C01810=1037.433,142.300,402.252,169.804,40.880,157.706
C01811=1037.427,142.051,402.274,169.802,40.880,157.706
C01812=1037.421,141.802,402.296,169.800,40.880,157.706
C01813=1037.415,141.552,402.317,169.797,40.880,157.706
C01814=1037.405,141.155,402.352,169.794,40.880,157.705
C01815=1037.395,140.757,402.386,169.790,40.881,157.705
C01816=1037.385,140.358,402.420,169.787,40.880,157.705
C01817=1037.376,139.961,402.454,169.783,40.880,157.705
C01818=1037.370,139.712,402.475,169.781,40.880,157.705
C01819=1037.363,139.462,402.497,169.777,40.880,157.704
C01820=1037.358,139.214,402.518,169.775,40.880,157.704
C01821=1037.352,138.965,402.540,169.773,40.880,157.704
C01822=1037.345,138.716,402.561,169.771,40.880,157.704
C01823=1037.339,138.467,402.583,169.768,40.880,157.704
C01824=1037.333,138.218,402.604,169.766,40.880,157.704
C01825=1037.327,137.968,402.625,169.764,40.880,157.704
C01826=1037.320,137.719,402.646,169.761,40.880,157.704
C01827=1037.315,137.471,402.667,169.759,40.880,157.704
C01828=1037.309,137.222,402.689,169.757,40.880,157.704
C01829=1037.302,136.973,402.710,169.754,40.880,157.703
C01830=1037.296,136.724,402.731,169.751,40.880,157.703
C01831=1037.290,136.474,402.752,169.749,40.881,157.703
C01832=1037.284,136.225,402.774,169.747,40.880,157.703
C01833=1037.277,135.976,402.795,169.744,40.881,157.703
C01834=1037.268,135.591,402.827,169.741,40.880,157.703
C01835=1037.259,135.205,402.861,169.737,40.881,157.703
C01836=1037.249,134.820,402.893,169.734,40.880,157.702
C01837=1037.240,134.434,402.925,169.730,40.881,157.702
C01838=1037.234,134.185,402.947,169.727,40.880,157.702
C01839=1037.227,133.936,402.968,169.725,40.881,157.702
C01840=1037.221,133.687,402.989,169.723,40.881,157.702
C01841=1037.215,133.438,403.010,169.720,40.881,157.702
C01842=1037.209,133.189,403.031,169.718,40.881,157.702
C01843=1037.203,132.940,403.052,169.716,40.881,157.702
C01844=1037.196,132.691,403.073,169.714,40.881,157.701
C01845=1037.190,132.441,403.094,169.711,40.881,157.701
C01846=1037.185,132.193,403.116,169.709,40.881,157.701
C01847=1037.178,131.943,403.136,169.707,40.881,157.701
C01848=1037.172,131.695,403.157,169.705,40.881,157.701
C01849=1037.166,131.446,403.179,169.703,40.881,157.701
C01850=1037.160,131.196,403.199,169.700,40.881,157.701
C01851=1037.154,130.948,403.220,169.698,40.881,157.701
C01852=1037.148,130.698,403.241,169.696,40.881,157.701
C01853=1037.141,130.449,403.262,169.693,40.881,157.700
C01854=1037.135,130.200,403.282,169.690,40.881,157.700
C01855=1037.129,129.951,403.303,169.688,40.882,157.700
C01856=1037.123,129.702,403.324,169.686,40.882,157.700
C01857=1037.116,129.453,403.345,169.683,40.882,157.700
C01858=1037.110,129.204,403.365,169.681,40.882,157.700
C01859=1037.104,128.955,403.387,169.679,40.882,157.700
C01860=1037.098,128.706,403.407,169.677,40.882,157.700
C01861=1037.091,128.457,403.428,169.674,40.883,157.700
C01862=1037.085,128.208,403.448,169.672,40.883,157.700
C01863=1037.079,127.958,403.469,169.670,40.883,157.700
C01864=1037.073,127.710,403.489,169.668,40.883,157.700
C01865=1037.067,127.460,403.510,169.665,40.883,157.699
C01866=1037.060,127.211,403.531,169.663,40.883,157.699
C01867=1037.054,126.962,403.551,169.661,40.884,157.699
C01868=1037.048,126.713,403.573,169.659,40.884,157.699
C01869=1037.042,126.464,403.593,169.655,40.883,157.699
C01870=1037.035,126.215,403.613,169.653,40.884,157.699
C01871=1037.029,125.967,403.634,169.651,40.884,157.699
C01872=1037.023,125.717,403.655,169.649,40.884,157.699
C01873=1037.016,125.467,403.675,169.646,40.884,157.699
C01874=1037.009,125.182,403.699,169.644,40.884,157.699
C01875=1037.002,124.897,403.723,169.641,40.884,157.699
C01876=1036.995,124.611,403.746,169.639,40.885,157.698
C01877=1036.988,124.325,403.770,169.636,40.885,157.698
C01878=1036.982,124.076,403.790,169.634,40.885,157.698
C01879=1036.976,123.826,403.811,169.632,40.885,157.698
C01880=1036.970,123.578,403.832,169.630,40.885,157.698
C01881=1036.963,123.329,403.852,169.627,40.885,157.698
C01882=1036.958,123.080,403.873,169.625,40.885,157.698
C01883=1036.951,122.831,403.894,169.623,40.885,157.698
C01884=1036.945,122.582,403.914,169.621,40.885,157.698
C01885=1036.938,122.332,403.934,169.619,40.886,157.698
C01886=1036.933,122.083,403.955,169.616,40.886,157.698
C01887=1036.926,121.834,403.976,169.613,40.886,157.697
C01888=1036.920,121.586,403.996,169.611,40.886,157.697
C01889=1036.914,121.336,404.016,169.609,40.886,157.697
C01890=1036.908,121.087,404.036,169.607,40.886,157.697
C01891=1036.902,120.839,404.057,169.604,40.886,157.697
C01892=1036.895,120.589,404.077,169.602,40.886,157.697
C01893=1036.890,120.340,404.098,169.600,40.886,157.697
C01894=1036.883,120.091,404.118,169.598,40.887,157.697
C01895=1036.877,119.842,404.138,169.596,40.887,157.697
C01896=1036.871,119.593,404.159,169.593,40.887,157.697
C01897=1036.865,119.344,404.180,169.591,40.887,157.696
C01898=1036.859,119.094,404.200,169.589,40.887,157.696
C01899=1036.853,118.845,404.220,169.587,40.887,157.696
C01900=1036.847,118.596,404.241,169.585,40.887,157.696
C01901=1036.841,118.347,404.261,169.581,40.887,157.696
C01902=1036.835,118.098,404.281,169.579,40.888,157.696
C01903=1036.828,117.849,404.302,169.577,40.888,157.696
C01904=1036.823,117.600,404.323,169.575,40.887,157.696
C01905=1036.817,117.351,404.343,169.573,40.888,157.696
C01906=1036.810,117.102,404.363,169.571,40.888,157.696
C01907=1036.804,116.853,404.383,169.568,40.888,157.696
C01908=1036.798,116.603,404.404,169.566,40.888,157.695
C01909=1036.792,116.354,404.424,169.564,40.888,157.695
C01910=1036.786,116.105,404.444,169.562,40.888,157.695
C01911=1036.780,115.856,404.464,169.560,40.888,157.695
C01912=1036.774,115.607,404.485,169.558,40.888,157.695
C01913=1036.768,115.358,404.504,169.556,40.888,157.695
C01914=1036.762,115.109,404.526,169.553,40.889,157.695
C01915=1036.756,114.860,404.545,169.550,40.888,157.695
C01916=1036.750,114.611,404.566,169.548,40.888,157.695
C01917=1036.744,114.362,404.586,169.546,40.889,157.695
C01918=1036.738,114.113,404.606,169.544,40.889,157.695
C01919=1036.732,113.864,404.626,169.542,40.888,157.694
C01920=1036.726,113.614,404.647,169.540,40.889,157.694
C01921=1036.720,113.365,404.667,169.537,40.889,157.694
C01922=1036.714,113.117,404.687,169.535,40.889,157.694
C01923=1036.707,112.867,404.707,169.533,40.889,157.694
C01924=1036.702,112.618,404.727,169.531,40.889,157.694
C01925=1036.696,112.369,404.747,169.529,40.889,157.694
C01926=1036.689,112.119,404.767,169.527,40.890,157.694
C01927=1036.683,111.870,404.787,169.524,40.890,157.694
C01928=1036.677,111.622,404.807,169.522,40.890,157.694
C01929=1036.670,111.372,404.827,169.520,40.890,157.694
C01930=1036.664,111.123,404.847,169.518,40.891,157.694
C01931=1036.659,110.874,404.866,169.516,40.890,157.693
C01932=1036.652,110.624,404.887,169.514,40.890,157.693
C01933=1036.646,110.376,404.907,169.511,40.891,157.693
C01934=1036.640,110.127,404.927,169.509,40.891,157.693
C01935=1036.633,109.878,404.946,169.507,40.891,157.693
C01936=1036.627,109.628,404.966,169.504,40.891,157.693
C01937=1036.621,109.379,404.986,169.502,40.892,157.693
C01938=1036.613,109.093,405.008,169.499,40.892,157.693
C01939=1036.606,108.807,405.031,169.497,40.892,157.693
C01940=1036.599,108.521,405.054,169.494,40.893,157.693
C01941=1036.592,108.236,405.077,169.492,40.893,157.693
C01942=1036.586,107.986,405.096,169.489,40.893,157.693
C01943=1036.579,107.738,405.116,169.487,40.893,157.693
C01944=1036.573,107.488,405.136,169.485,40.893,157.692
C01945=1036.567,107.239,405.155,169.483,40.893,157.692
C01946=1036.561,106.990,405.175,169.481,40.893,157.692
C01947=1036.555,106.741,405.195,169.479,40.894,157.692
C01948=1036.548,106.491,405.214,169.476,40.894,157.692
C01949=1036.542,106.243,405.234,169.474,40.894,157.692
C01950=1036.536,105.994,405.254,169.472,40.894,157.692
C01951=1036.530,105.744,405.274,169.470,40.895,157.692
C01952=1036.524,105.495,405.294,169.468,40.895,157.692
C01953=1036.517,105.246,405.313,169.466,40.895,157.692
C01954=1036.512,104.997,405.332,169.463,40.896,157.692
C01955=1036.505,104.747,405.353,169.461,40.896,157.692
C01956=1036.499,104.499,405.373,169.459,40.895,157.691
C01957=1036.493,104.249,405.392,169.457,40.896,157.691
C01958=1036.486,104.001,405.411,169.455,40.896,157.691
C01959=1036.481,103.751,405.431,169.453,40.896,157.691
C01960=1036.474,103.502,405.451,169.451,40.896,157.691
C01961=1036.468,103.253,405.471,169.448,40.897,157.691
C01962=1036.463,103.003,405.490,169.446,40.897,157.691
C01963=1036.456,102.755,405.509,169.443,40.897,157.691
C01964=1036.450,102.505,405.529,169.441,40.897,157.691
C01965=1036.444,102.256,405.549,169.439,40.897,157.691
C01966=1036.438,102.007,405.568,169.437,40.897,157.691
C01967=1036.432,101.758,405.588,169.435,40.897,157.691
C01968=1036.425,101.509,405.608,169.433,40.898,157.691
C01969=1036.419,101.260,405.627,169.430,40.898,157.691
C01970=1036.413,101.010,405.647,169.428,40.898,157.691
C01971=1036.407,100.761,405.666,169.426,40.898,157.690
C01972=1036.400,100.512,405.686,169.424,40.899,157.690
C01973=1036.395,100.263,405.705,169.422,40.898,157.690
C01974=1036.389,100.014,405.725,169.420,40.898,157.690
C01975=1036.382,99.765,405.744,169.418,40.899,157.690
C01976=1036.376,99.515,405.763,169.415,40.900,157.690
C01977=1036.369,99.266,405.783,169.413,40.900,157.690
C01978=1036.364,99.017,405.802,169.411,40.900,157.690
C01979=1036.357,98.768,405.821,169.409,40.900,157.690
C01980=1036.351,98.519,405.840,169.407,40.901,157.690
C01981=1036.344,98.269,405.859,169.405,40.901,157.690
C01982=1036.338,98.020,405.879,169.402,40.901,157.690
C01983=1036.332,97.771,405.898,169.400,40.901,157.690
C01984=1036.326,97.522,405.917,169.398,40.902,157.690
C01985=1036.319,97.273,405.937,169.396,40.902,157.690
C01986=1036.314,97.024,405.956,169.394,40.902,157.690
C01987=1036.307,96.774,405.975,169.392,40.902,157.689
C01988=1036.301,96.525,405.995,169.390,40.903,157.689
C01989=1036.294,96.276,406.014,169.387,40.903,157.689
C01990=1036.288,96.027,406.033,169.385,40.903,157.689
C01991=1036.282,95.778,406.052,169.383,40.903,157.689
C01992=1036.276,95.529,406.071,169.381,40.904,157.689
C01993=1036.270,95.280,406.090,169.379,40.904,157.689
C01994=1036.264,95.030,406.109,169.376,40.903,157.689
C01995=1036.257,94.781,406.129,169.374,40.904,157.689
C01996=1036.251,94.532,406.148,169.371,40.904,157.689
C01997=1036.244,94.282,406.167,169.369,40.904,157.689
C01998=1036.239,94.033,406.186,169.367,40.904,157.689
C01999=1036.232,93.785,406.206,169.365,40.905,157.689
C02000=1036.226,93.535,406.225,169.363,40.905,157.689
C02001=1036.220,93.286,406.243,169.361,40.905,157.688
C02002=1036.213,93.000,406.266,169.358,40.905,157.688
C02003=1036.205,92.714,406.287,169.356,40.906,157.688
C02004=1036.199,92.429,406.310,169.353,40.906,157.688
C02005=1036.192,92.142,406.332,169.351,40.906,157.688
C02006=1036.186,91.893,406.350,169.349,40.907,157.688
C02007=1036.180,91.644,406.369,169.347,40.907,157.688
C02008=1036.173,91.395,406.389,169.345,40.907,157.688
C02009=1036.168,91.146,406.408,169.343,40.907,157.688
C02010=1036.161,90.897,406.427,169.340,40.908,157.688
C02011=1036.155,90.648,406.445,169.338,40.908,157.688
C02012=1036.149,90.398,406.465,169.336,40.908,157.688
C02013=1036.143,90.149,406.483,169.334,40.908,157.688
C02014=1036.137,89.900,406.503,169.332,40.908,157.688
C02015=1036.130,89.651,406.522,169.330,40.909,157.688
C02016=1036.123,89.401,406.541,169.328,40.909,157.688
C02017=1036.117,89.152,406.560,169.325,40.909,157.687
C02018=1036.111,88.903,406.579,169.323,40.910,157.687
C02019=1036.105,88.654,406.597,169.321,40.910,157.687
C02020=1036.098,88.404,406.616,169.319,40.910,157.687
C02021=1036.092,88.155,406.635,169.317,40.910,157.687
C02022=1036.085,87.906,406.653,169.315,40.910,157.687
C02023=1036.080,87.657,406.673,169.313,40.911,157.687
C02024=1036.073,87.408,406.691,169.310,40.912,157.687
C02025=1036.067,87.159,406.710,169.308,40.912,157.687
C02026=1036.060,86.909,406.729,169.306,40.912,157.687
C02027=1036.054,86.660,406.747,169.304,40.912,157.687
C02028=1036.048,86.411,406.766,169.302,40.913,157.687
C02029=1036.042,86.161,406.784,169.300,40.913,157.687
C02030=1036.036,85.912,406.803,169.298,40.913,157.687
C02031=1036.029,85.663,406.822,169.295,40.913,157.687
C02032=1036.023,85.414,406.840,169.293,40.914,157.687
C02033=1036.017,85.164,406.860,169.291,40.914,157.687
C02034=1036.011,84.915,406.878,169.289,40.914,157.687
C02035=1036.004,84.666,406.897,169.286,40.914,157.686
C02036=1035.998,84.417,406.916,169.284,40.915,157.686
C02037=1035.992,84.168,406.934,169.282,40.915,157.686
C02038=1035.985,83.919,406.953,169.279,40.915,157.686
C02039=1035.979,83.669,406.972,169.278,40.916,157.686
C02040=1035.973,83.420,406.990,169.276,40.916,157.686
C02041=1035.967,83.170,407.009,169.273,40.916,157.686
C02042=1035.960,82.921,407.027,169.271,40.917,157.686
C02043=1035.954,82.672,407.046,169.269,40.917,157.686
C02044=1035.948,82.423,407.065,169.267,40.917,157.686
C02045=1035.942,82.174,407.084,169.265,40.917,157.686
C02046=1035.936,81.925,407.102,169.262,40.918,157.686
C02047=1035.930,81.675,407.120,169.260,40.918,157.686
C02048=1035.924,81.426,407.139,169.258,40.918,157.686
C02049=1035.917,81.177,407.157,169.256,40.918,157.686
C02050=1035.911,80.928,407.176,169.254,40.919,157.686
C02051=1035.905,80.679,407.195,169.252,40.919,157.686
C02052=1035.899,80.429,407.213,169.250,40.919,157.686
C02053=1035.892,80.180,407.232,169.248,40.919,157.686
C02054=1035.886,79.931,407.250,169.246,40.920,157.685
C02055=1035.880,79.682,407.269,169.243,40.920,157.685
C02056=1035.874,79.432,407.287,169.241,40.920,157.685
C02057=1035.868,79.183,407.306,169.239,40.920,157.685
C02058=1035.862,78.934,407.325,169.237,40.921,157.685
C02059=1035.856,78.685,407.343,169.235,40.921,157.685
C02060=1035.849,78.435,407.361,169.233,40.921,157.685
C02061=1035.843,78.186,407.380,169.231,40.921,157.685
C02062=1035.837,77.937,407.398,169.229,40.922,157.685
C02063=1035.830,77.687,407.416,169.226,40.922,157.685
C02064=1035.824,77.438,407.435,169.224,40.922,157.685
C02065=1035.818,77.190,407.453,169.222,40.922,157.685
C02066=1035.811,76.903,407.475,169.220,40.923,157.685
C02067=1035.804,76.617,407.495,169.217,40.924,157.685
C02068=1035.796,76.331,407.516,169.215,40.924,157.685
C02069=1035.790,76.046,407.537,169.212,40.924,157.685
C02070=1035.783,75.797,407.556,169.210,40.924,157.685
C02071=1035.777,75.547,407.574,169.208,40.925,157.684
C02072=1035.771,75.298,407.592,169.206,40.925,157.684
C02073=1035.764,75.048,407.610,169.204,40.925,157.684
C02074=1035.757,74.799,407.628,169.202,40.925,157.684
C02075=1035.751,74.549,407.646,169.200,40.926,157.684
C02076=1035.745,74.301,407.665,169.197,40.927,157.684
C02077=1035.739,74.051,407.683,169.195,40.927,157.684
C02078=1035.733,73.802,407.701,169.193,40.927,157.684
C02079=1035.727,73.553,407.720,169.191,40.927,157.684
C02080=1035.720,73.303,407.738,169.189,40.928,157.684
C02081=1035.713,73.054,407.756,169.187,40.928,157.684
C02082=1035.708,72.805,407.773,169.185,40.928,157.684
C02083=1035.701,72.556,407.792,169.182,40.928,157.684
C02084=1035.695,72.307,407.810,169.180,40.929,157.684
C02085=1035.689,72.057,407.829,169.178,40.929,157.684
C02086=1035.683,71.808,407.847,169.176,40.930,157.684
C02087=1035.677,71.559,407.864,169.174,40.930,157.684
C02088=1035.671,71.309,407.883,169.172,40.930,157.684
C02089=1035.664,71.060,407.900,169.170,40.930,157.684
C02090=1035.657,70.811,407.919,169.168,40.931,157.684
C02091=1035.651,70.561,407.937,169.165,40.931,157.683
C02092=1035.645,70.313,407.955,169.163,40.931,157.683
C02093=1035.639,70.063,407.973,169.161,40.931,157.683
C02094=1035.633,69.813,407.991,169.159,40.932,157.683
C02095=1035.626,69.564,408.009,169.157,40.933,157.683
C02096=1035.621,69.315,408.026,169.155,40.933,157.683
C02097=1035.614,69.066,408.045,169.153,40.933,157.683
C02098=1035.608,68.817,408.063,169.150,40.933,157.683
C02099=1035.601,68.567,408.080,169.148,40.934,157.683
C02100=1035.595,68.318,408.099,169.146,40.934,157.683
C02101=1035.589,68.069,408.117,169.144,40.934,157.683
C02102=1035.583,67.819,408.135,169.142,40.934,157.683
C02103=1035.576,67.570,408.153,169.140,40.935,157.683
C02104=1035.570,67.321,408.171,169.138,40.935,157.683
C02105=1035.564,67.072,408.188,169.135,40.936,157.683
C02106=1035.557,66.822,408.205,169.133,40.936,157.683
C02107=1035.551,66.573,408.224,169.131,40.936,157.683
C02108=1035.545,66.324,408.242,169.129,40.936,157.683
C02109=1035.539,66.075,408.259,169.127,40.937,157.683
C02110=1035.532,65.826,408.278,169.125,40.938,157.683
C02111=1035.526,65.576,408.296,169.123,40.938,157.683
C02112=1035.520,65.327,408.313,169.120,40.938,157.683
C02113=1035.514,65.077,408.330,169.118,40.938,157.683
C02114=1035.508,64.828,408.348,169.116,40.939,157.682
C02115=1035.501,64.579,408.366,169.114,40.939,157.682
C02116=1035.495,64.330,408.384,169.112,40.940,157.682
C02117=1035.488,64.080,408.401,169.110,40.940,157.682
C02118=1035.482,63.831,408.419,169.108,40.940,157.682
C02119=1035.476,63.581,408.437,169.105,40.940,157.682
C02120=1035.470,63.332,408.454,169.103,40.941,157.682
C02121=1035.462,63.083,408.472,169.101,40.942,157.682
C02122=1035.456,62.834,408.490,169.099,40.942,157.682
C02123=1035.450,62.585,408.507,169.097,40.942,157.682
C02124=1035.444,62.335,408.525,169.095,40.943,157.682
C02125=1035.437,62.086,408.542,169.092,40.943,157.682
C02126=1035.431,61.837,408.559,169.090,40.944,157.682
C02127=1035.425,61.587,408.577,169.088,40.944,157.682
C02128=1035.418,61.338,408.595,169.086,40.945,157.682
C02129=1035.411,61.088,408.612,169.084,40.945,157.682
C02130=1035.404,60.802,408.632,169.081,40.945,157.682
C02131=1035.397,60.516,408.652,169.079,40.946,157.682
C02132=1035.389,60.230,408.672,169.076,40.946,157.682
C02133=1035.382,59.944,408.692,169.074,40.947,157.682
C02134=1035.376,59.694,408.710,169.071,40.948,157.682
C02135=1035.369,59.446,408.727,169.069,40.948,157.682
C02136=1035.363,59.196,408.744,169.067,40.948,157.682
C02137=1035.356,58.947,408.762,169.065,40.948,157.682
C02138=1035.350,58.698,408.779,169.063,40.949,157.682
C02139=1035.344,58.448,408.797,169.060,40.950,157.682
C02140=1035.337,58.199,408.814,169.058,40.950,157.682
C02141=1035.331,57.950,408.831,169.056,40.950,157.682
C02142=1035.325,57.700,408.849,169.054,40.951,157.682
C02143=1035.318,57.451,408.866,169.052,40.951,157.682
C02144=1035.312,57.202,408.883,169.050,40.951,157.682
C02145=1035.305,56.952,408.901,169.047,40.952,157.681
C02146=1035.299,56.703,408.919,169.045,40.953,157.682
C02147=1035.292,56.454,408.935,169.043,40.953,157.681
C02148=1035.286,56.204,408.953,169.041,40.953,157.681
C02149=1035.280,55.956,408.970,169.039,40.953,157.681
C02150=1035.273,55.706,408.988,169.037,40.954,157.681
C02151=1035.267,55.456,409.005,169.034,40.955,157.681
C02152=1035.261,55.207,409.022,169.032,40.955,157.681
C02153=1035.254,54.958,409.039,169.030,40.955,157.681
C02154=1035.249,54.709,409.057,169.028,40.955,157.681
C02155=1035.242,54.459,409.074,169.026,40.956,157.681
C02156=1035.236,54.210,409.091,169.024,40.956,157.681
C02157=1035.229,53.961,409.109,169.021,40.957,157.681
C02158=1035.223,53.711,409.126,169.019,40.957,157.681
C02159=1035.217,53.462,409.143,169.017,40.957,157.681
C02160=1035.211,53.212,409.161,169.015,40.958,157.681
C02161=1035.204,52.963,409.178,169.013,40.958,157.681
C02162=1035.197,52.714,409.195,169.011,40.959,157.681
C02163=1035.192,52.464,409.212,169.008,40.959,157.681
C02164=1035.185,52.215,409.229,169.006,40.959,157.681
C02165=1035.179,51.966,409.246,169.004,40.960,157.681
C02166=1035.173,51.716,409.264,169.002,40.960,157.681
C02167=1035.167,51.468,409.281,169.000,40.960,157.681
C02168=1035.160,51.218,409.298,168.998,40.961,157.681
C02169=1035.155,50.969,409.315,168.995,40.961,157.681
C02170=1035.148,50.719,409.332,168.993,40.962,157.681
C02171=1035.142,50.471,409.349,168.991,40.962,157.681
C02172=1035.135,50.220,409.366,168.989,40.962,157.681
C02173=1035.129,49.971,409.384,168.987,40.963,157.680
C02174=1035.123,49.722,409.401,168.985,40.963,157.680
C02175=1035.116,49.473,409.418,168.982,40.963,157.680
C02176=1035.111,49.223,409.435,168.980,40.964,157.680
C02177=1035.104,48.974,409.452,168.978,40.964,157.680
C02178=1035.097,48.725,409.469,168.976,40.965,157.680
C02179=1035.092,48.475,409.486,168.974,40.965,157.680
C02180=1035.085,48.226,409.504,168.972,40.965,157.680
C02181=1035.079,47.977,409.521,168.969,40.965,157.680
C02182=1035.073,47.727,409.537,168.967,40.966,157.680
C02183=1035.067,47.478,409.555,168.965,40.966,157.680
C02184=1035.061,47.229,409.572,168.963,40.967,157.680
C02185=1035.054,46.979,409.588,168.961,40.967,157.680
C02186=1035.049,46.730,409.606,168.959,40.967,157.680
C02187=1035.042,46.481,409.623,168.957,40.967,157.680
C02188=1035.036,46.231,409.640,168.954,40.968,157.680
C02189=1035.029,45.982,409.657,168.952,40.969,157.680
C02190=1035.024,45.732,409.674,168.950,40.969,157.680
C02191=1035.018,45.483,409.691,168.948,40.969,157.680
C02192=1035.011,45.234,409.708,168.946,40.969,157.680
C02193=1035.005,44.985,409.724,168.944,40.970,157.680
C02194=1034.998,44.699,409.744,168.941,40.970,157.679
C02195=1034.991,44.411,409.764,168.939,40.970,157.679
C02196=1034.984,44.125,409.783,168.936,40.971,157.679
C02197=1034.977,43.839,409.803,168.934,40.971,157.679
C02198=1034.971,43.590,409.819,168.932,40.972,157.679
C02199=1034.964,43.340,409.837,168.929,40.972,157.679
C02200=1034.958,43.091,409.853,168.927,40.972,157.679
C02201=1034.951,42.841,409.870,168.925,40.972,157.679
C02202=1034.945,42.592,409.887,168.923,40.973,157.679
C02203=1034.940,42.343,409.904,168.921,40.974,157.679
C02204=1034.933,42.093,409.921,168.918,40.974,157.679
C02205=1034.927,41.844,409.938,168.916,40.974,157.679
C02206=1034.920,41.594,409.954,168.914,40.975,157.679
C02207=1034.914,41.345,409.971,168.912,40.975,157.679
C02208=1034.908,41.096,409.988,168.910,40.975,157.679
C02209=1034.902,40.846,410.004,168.907,40.976,157.679
C02210=1034.895,40.597,410.021,168.905,40.977,157.679
C02211=1034.889,40.348,410.037,168.903,40.977,157.679
C02212=1034.883,40.098,410.054,168.901,40.977,157.679
C02213=1034.877,39.849,410.071,168.899,40.977,157.679
C02214=1034.870,39.599,410.088,168.896,40.978,157.679
C02215=1034.864,39.350,410.105,168.894,40.979,157.679
C02216=1034.858,39.101,410.121,168.892,40.979,157.679
C02217=1034.851,38.851,410.137,168.890,40.979,157.679
C02218=1034.845,38.602,410.154,168.888,40.979,157.679
C02219=1034.839,38.353,410.171,168.886,40.980,157.679
C02220=1034.833,38.103,410.187,168.883,40.981,157.679
C02221=1034.826,37.854,410.204,168.881,40.981,157.678
C02222=1034.820,37.605,410.221,168.879,40.981,157.678
C02223=1034.814,37.355,410.237,168.877,40.982,157.678
C02224=1034.807,37.106,410.253,168.875,40.982,157.678
C02225=1034.801,36.857,410.270,168.872,40.982,157.678
C02226=1034.794,36.607,410.286,168.870,40.983,157.678
C02227=1034.788,36.358,410.303,168.868,40.984,157.678
C02228=1034.782,36.108,410.319,168.866,40.984,157.678
C02229=1034.775,35.858,410.335,168.863,40.985,157.678
C02230=1034.769,35.610,410.352,168.861,40.985,157.678
C02231=1034.763,35.360,410.368,168.859,40.985,157.678
C02232=1034.757,35.111,410.384,168.858,40.986,157.678
C02233=1034.750,34.861,410.400,168.855,40.987,157.678
C02234=1034.744,34.612,410.417,168.853,40.987,157.678
C02235=1034.737,34.363,410.434,168.851,40.988,157.678
C02236=1034.731,34.113,410.450,168.849,40.988,157.678
C02237=1034.724,33.864,410.466,168.846,40.988,157.678
C02238=1034.718,33.615,410.482,168.844,40.989,157.678
C02239=1034.712,33.365,410.499,168.842,40.989,157.678
C02240=1034.706,33.115,410.515,168.840,40.990,157.678
C02241=1034.700,32.866,410.531,168.838,40.990,157.678
C02242=1034.693,32.617,410.547,168.835,40.991,157.678
C02243=1034.686,32.368,410.564,168.833,40.991,157.678
C02244=1034.680,32.118,410.581,168.831,40.991,157.678
C02245=1034.674,31.869,410.597,168.829,40.992,157.678
C02246=1034.668,31.620,410.613,168.826,40.993,157.678
C02247=1034.662,31.371,410.629,168.824,40.993,157.678
C02248=1034.655,31.120,410.645,168.822,40.994,157.678
C02249=1034.649,30.871,410.662,168.820,40.994,157.678
C02250=1034.643,30.622,410.677,168.817,40.994,157.678
C02251=1034.637,30.373,410.694,168.815,40.995,157.678
C02252=1034.630,30.123,410.710,168.813,40.995,157.678
C02253=1034.623,29.874,410.726,168.811,40.996,157.678
C02254=1034.617,29.624,410.742,168.808,40.996,157.678
C02255=1034.611,29.375,410.758,168.806,40.997,157.678
C02256=1034.606,29.126,410.775,168.804,40.997,157.678
C02257=1034.598,28.876,410.791,168.802,40.997,157.677
C02258=1034.592,28.589,410.810,168.799,40.998,157.678
C02259=1034.584,28.303,410.829,168.797,40.999,157.677
C02260=1034.577,28.016,410.847,168.794,40.999,157.677
C02261=1034.570,27.730,410.865,168.791,41.000,157.677
C02262=1034.563,27.481,410.881,168.789,41.000,157.677
C02263=1034.557,27.232,410.897,168.787,41.000,157.677
C02264=1034.551,26.982,410.913,168.785,41.001,157.677
C02265=1034.544,26.733,410.929,168.782,41.002,157.677
C02266=1034.538,26.483,410.946,168.780,41.002,157.677
C02267=1034.531,26.233,410.961,168.778,41.003,157.677
C02268=1034.526,25.984,410.977,168.776,41.003,157.677
C02269=1034.519,25.735,410.992,168.773,41.004,157.677
C02270=1034.513,25.486,411.009,168.771,41.004,157.677
C02271=1034.506,25.237,411.024,168.769,41.004,157.677
C02272=1034.500,24.987,411.041,168.767,41.005,157.677
C02273=1034.493,24.737,411.056,168.764,41.006,157.677
C02274=1034.487,24.488,411.072,168.762,41.006,157.677
C02275=1034.481,24.239,411.088,168.761,41.007,157.677
C02276=1034.475,23.989,411.104,168.758,41.007,157.677
C02277=1034.468,23.740,411.120,168.756,41.008,157.677
C02278=1034.462,23.490,411.136,168.754,41.008,157.677
C02279=1034.455,23.241,411.151,168.752,41.008,157.677
C02280=1034.449,22.991,411.168,168.749,41.009,157.677
C02281=1034.442,22.742,411.183,168.747,41.010,157.677
C02282=1034.436,22.493,411.200,168.745,41.010,157.677
C02283=1034.430,22.243,411.214,168.743,41.011,157.677
C02284=1034.424,21.994,411.231,168.740,41.011,157.677
C02285=1034.417,21.745,411.246,168.738,41.011,157.677
C02286=1034.411,21.495,411.263,168.736,41.012,157.677
C02287=1034.405,21.246,411.278,168.733,41.013,157.677
C02288=1034.399,20.996,411.294,168.731,41.014,157.677
C02289=1034.392,20.747,411.310,168.729,41.014,157.677
C02290=1034.386,20.497,411.325,168.727,41.014,157.677
C02291=1034.380,20.248,411.341,168.724,41.015,157.677
C02292=1034.374,19.998,411.357,168.722,41.015,157.677
C02293=1034.367,19.749,411.372,168.720,41.015,157.677
C02294=1034.361,19.499,411.389,168.717,41.016,157.677
C02295=1034.355,19.250,411.404,168.715,41.017,157.677
C02296=1034.348,19.001,411.419,168.713,41.017,157.677
C02297=1034.342,18.751,411.435,168.711,41.018,157.677
C02298=1034.336,18.502,411.451,168.708,41.018,157.677
C02299=1034.329,18.253,411.466,168.706,41.019,157.677
C02300=1034.323,18.003,411.482,168.704,41.019,157.677
C02301=1034.317,17.754,411.497,168.701,41.020,157.677
C02302=1034.310,17.505,411.513,168.699,41.021,157.676
C02303=1034.304,17.255,411.528,168.697,41.021,157.676
C02304=1034.298,17.006,411.544,168.694,41.022,157.676
C02305=1034.290,16.756,411.560,168.692,41.022,157.676
C02306=1034.285,16.506,411.576,168.691,41.023,157.676
C02307=1034.278,16.257,411.591,168.688,41.023,157.676
C02308=1034.272,16.007,411.606,168.685,41.024,157.676
C02309=1034.266,15.758,411.623,168.684,41.024,157.676
C02310=1034.259,15.508,411.637,168.682,41.025,157.676
C02311=1034.253,15.259,411.653,168.679,41.025,157.676
C02312=1034.247,15.009,411.669,168.677,41.026,157.676
C02313=1034.240,14.760,411.684,168.675,41.026,157.676
C02314=1034.234,14.510,411.699,168.672,41.027,157.676
C02315=1034.228,14.261,411.716,168.670,41.027,157.676
C02316=1034.222,14.011,411.730,168.668,41.028,157.676
C02317=1034.215,13.762,411.746,168.665,41.029,157.676
C02318=1034.209,13.513,411.761,168.663,41.029,157.676
C02319=1034.202,13.263,411.776,168.661,41.030,157.676
C02320=1034.196,13.014,411.792,168.658,41.030,157.676
C02321=1034.190,12.764,411.807,168.656,41.031,157.676
C02322=1034.183,12.480,411.825,168.653,41.032,157.676
C02323=1034.175,12.194,411.842,168.651,41.032,157.676
C02324=1034.168,11.908,411.859,168.648,41.033,157.676
C02325=1034.161,11.623,411.877,168.645,41.034,157.676
C02326=1034.154,11.374,411.892,168.643,41.034,157.676
C02327=1034.148,11.125,411.907,168.640,41.035,157.676
C02328=1034.141,10.875,411.922,168.638,41.036,157.676
C02329=1034.135,10.625,411.937,168.636,41.036,157.676
C02330=1034.128,10.376,411.953,168.634,41.037,157.676
C02331=1034.122,10.127,411.968,168.632,41.037,157.676
C02332=1034.115,9.877,411.983,168.630,41.038,157.676
C02333=1034.109,9.629,411.998,168.627,41.038,157.676
C02334=1034.103,9.379,412.013,168.625,41.039,157.676
C02335=1034.097,9.129,412.028,168.623,41.040,157.676
C02336=1034.090,8.880,412.043,168.620,41.041,157.676
C02337=1034.083,8.631,412.059,168.618,41.041,157.676
C02338=1034.077,8.381,412.074,168.615,41.042,157.676
C02339=1034.071,8.131,412.089,168.613,41.042,157.676
C02340=1034.064,7.882,412.104,168.611,41.043,157.676
C02341=1034.058,7.632,412.119,168.608,41.043,157.676
C02342=1034.051,7.383,412.134,168.606,41.044,157.676
C02343=1034.045,7.133,412.149,168.604,41.044,157.676
C02344=1034.040,6.884,412.164,168.601,41.045,157.676
C02345=1034.033,6.634,412.179,168.599,41.046,157.676
C02346=1034.027,6.385,412.194,168.597,41.047,157.676
C02347=1034.020,6.136,412.210,168.594,41.047,157.676
C02348=1034.014,5.886,412.225,168.592,41.048,157.676
C02349=1034.008,5.636,412.240,168.589,41.048,157.676
C02350=1034.001,5.387,412.255,168.588,41.049,157.676
C02351=1033.995,5.138,412.269,168.585,41.049,157.676
C02352=1033.989,4.888,412.284,168.583,41.050,157.676
C02353=1033.982,4.639,412.300,168.581,41.051,157.676
C02354=1033.976,4.389,412.315,168.579,41.051,157.676
C02355=1033.970,4.140,412.330,168.576,41.052,157.676
C02356=1033.963,3.890,412.345,168.574,41.053,157.676
C02357=1033.957,3.641,412.359,168.571,41.053,157.676
C02358=1033.951,3.391,412.374,168.569,41.053,157.676
C02359=1033.945,3.142,412.389,168.567,41.054,157.676
C02360=1033.938,2.892,412.404,168.564,41.054,157.676
C02361=1033.932,2.642,412.419,168.562,41.055,157.676
C02362=1033.926,2.393,412.434,168.560,41.056,157.676
C02363=1033.920,2.144,412.449,168.557,41.057,157.676
C02364=1033.913,1.894,412.464,168.555,41.057,157.676
C02365=1033.907,1.645,412.478,168.552,41.058,157.676
C02366=1033.900,1.395,412.494,168.550,41.058,157.676
C02367=1033.894,1.147,412.509,168.548,41.058,157.676
C02368=1033.888,0.897,412.524,168.545,41.059,157.676
C02369=1033.882,0.647,412.539,168.543,41.060,157.676
C02370=1033.875,0.398,412.554,168.541,41.060,157.676
C02371=1033.870,0.149,412.568,168.538,41.061,157.676
C02372=1033.863,-0.101,412.583,168.536,41.062,157.676
C02373=1033.857,-0.351,412.598,168.533,41.062,157.675
C02374=1033.850,-0.600,412.613,168.531,41.062,157.675
C02375=1033.845,-0.850,412.627,168.529,41.063,157.675
C02376=1033.839,-1.100,412.642,168.526,41.064,157.675
C02377=1033.832,-1.349,412.657,168.525,41.064,157.675
C02378=1033.826,-1.598,412.671,168.523,41.065,157.675
C02379=1033.820,-1.848,412.686,168.520,41.066,157.675
C02380=1033.814,-2.098,412.701,168.518,41.066,157.675
C02381=1033.807,-2.347,412.716,168.515,41.066,157.675
C02382=1033.801,-2.596,412.731,168.513,41.067,157.675
C02383=1033.795,-2.846,412.746,168.511,41.067,157.675
C02384=1033.789,-3.095,412.761,168.508,41.068,157.675
C02385=1033.783,-3.344,412.775,168.506,41.069,157.675
C02386=1033.776,-3.628,412.792,168.503,41.069,157.675
C02387=1033.769,-3.911,412.808,168.500,41.070,157.675
C02388=1033.761,-4.194,412.825,168.498,41.071,157.675
C02389=1033.754,-4.478,412.841,168.495,41.072,157.675
C02390=1033.747,-4.727,412.856,168.492,41.072,157.675
C02391=1033.741,-4.977,412.870,168.490,41.073,157.675
C02392=1033.735,-5.226,412.885,168.487,41.074,157.675
C02393=1033.728,-5.476,412.899,168.485,41.074,157.675
C02394=1033.722,-5.725,412.914,168.483,41.075,157.675
C02395=1033.716,-5.975,412.928,168.480,41.076,157.675
C02396=1033.709,-6.224,412.942,168.479,41.077,157.675
C02397=1033.703,-6.474,412.957,168.475,41.077,157.675
C02398=1033.697,-6.724,412.971,168.474,41.078,157.675
C02399=1033.690,-6.973,412.985,168.471,41.079,157.675
C02400=1033.684,-7.222,413.000,168.469,41.079,157.675
C02401=1033.678,-7.473,413.014,168.466,41.080,157.675
C02402=1033.671,-7.721,413.028,168.464,41.080,157.675
C02403=1033.665,-7.971,413.043,168.461,41.081,157.675
C02404=1033.659,-8.221,413.057,168.459,41.082,157.675
C02405=1033.652,-8.470,413.072,168.457,41.082,157.675
C02406=1033.646,-8.720,413.086,168.454,41.083,157.675
C02407=1033.640,-8.969,413.100,168.452,41.084,157.675
C02408=1033.633,-9.219,413.115,168.449,41.085,157.675
C02409=1033.627,-9.468,413.130,168.447,41.086,157.675
C02410=1033.621,-9.717,413.143,168.444,41.086,157.675
C02411=1033.614,-9.967,413.158,168.442,41.087,157.675
C02412=1033.609,-10.217,413.172,168.439,41.087,157.675
C02413=1033.602,-10.466,413.186,168.438,41.088,157.675
C02414=1033.595,-10.716,413.201,168.435,41.088,157.675
C02415=1033.589,-10.965,413.214,168.433,41.089,157.675
C02416=1033.583,-11.215,413.229,168.430,41.090,157.675
C02417=1033.577,-11.464,413.243,168.428,41.091,157.675
C02418=1033.570,-11.714,413.257,168.425,41.092,157.675
C02419=1033.565,-11.963,413.271,168.423,41.092,157.675
C02420=1033.558,-12.213,413.286,168.421,41.093,157.675
C02421=1033.551,-12.463,413.300,168.418,41.093,157.675
C02422=1033.546,-12.712,413.314,168.416,41.094,157.675
C02423=1033.539,-12.962,413.328,168.413,41.095,157.675
C02424=1033.533,-13.211,413.343,168.411,41.095,157.675
C02425=1033.527,-13.461,413.357,168.408,41.096,157.675
C02426=1033.520,-13.709,413.371,168.406,41.097,157.675
C02427=1033.514,-13.960,413.385,168.403,41.098,157.675
C02428=1033.508,-14.208,413.399,168.401,41.098,157.675
C02429=1033.502,-14.459,413.413,168.398,41.099,157.675
C02430=1033.496,-14.708,413.428,168.396,41.099,157.675
C02431=1033.489,-14.958,413.442,168.394,41.100,157.675
C02432=1033.484,-15.207,413.455,168.392,41.101,157.675
C02433=1033.477,-15.457,413.470,168.389,41.101,157.675
C02434=1033.471,-15.707,413.484,168.387,41.102,157.675
C02435=1033.464,-15.955,413.498,168.384,41.103,157.675
C02436=1033.457,-16.205,413.512,168.382,41.103,157.675
C02437=1033.452,-16.455,413.525,168.379,41.104,157.675
C02438=1033.445,-16.704,413.540,168.377,41.105,157.675
C02439=1033.439,-16.954,413.554,168.374,41.106,157.675
C02440=1033.432,-17.204,413.567,168.372,41.107,157.675
C02441=1033.426,-17.453,413.581,168.369,41.108,157.675
C02442=1033.420,-17.703,413.596,168.367,41.108,157.675
C02443=1033.413,-17.952,413.609,168.364,41.109,157.675
C02444=1033.407,-18.202,413.622,168.363,41.110,157.675
C02445=1033.401,-18.451,413.637,168.360,41.111,157.675
C02446=1033.394,-18.701,413.651,168.357,41.111,157.675
C02447=1033.388,-18.950,413.664,168.355,41.112,157.675
C02448=1033.382,-19.200,413.678,168.352,41.113,157.675
C02449=1033.375,-19.449,413.692,168.350,41.113,157.675
C02450=1033.369,-19.731,413.707,168.347,41.114,157.675
C02451=1033.361,-20.013,413.723,168.344,41.115,157.675
C02452=1033.354,-20.294,413.738,168.341,41.116,157.675
C02453=1033.347,-20.576,413.754,168.338,41.117,157.675
C02454=1033.341,-20.826,413.768,168.336,41.118,157.675
C02455=1033.334,-21.075,413.781,168.333,41.119,157.675
C02456=1033.328,-21.324,413.796,168.331,41.119,157.675
C02457=1033.322,-21.574,413.809,168.329,41.120,157.675
C02458=1033.315,-21.824,413.823,168.327,41.121,157.675
C02459=1033.310,-22.073,413.837,168.324,41.121,157.675
C02460=1033.303,-22.323,413.850,168.322,41.122,157.675
C02461=1033.297,-22.572,413.864,168.319,41.123,157.675
C02462=1033.291,-22.822,413.877,168.316,41.123,157.675
C02463=1033.284,-23.071,413.892,168.314,41.124,157.675
C02464=1033.278,-23.321,413.905,168.311,41.125,157.675
C02465=1033.272,-23.570,413.919,168.309,41.126,157.675
C02466=1033.266,-23.820,413.933,168.306,41.127,157.675
C02467=1033.259,-24.069,413.946,168.304,41.127,157.675
C02468=1033.253,-24.320,413.960,168.301,41.128,157.675
C02469=1033.247,-24.569,413.973,168.299,41.129,157.675
C02470=1033.241,-24.818,413.987,168.296,41.130,157.675
C02471=1033.234,-25.068,414.000,168.294,41.130,157.675
C02472=1033.228,-25.318,414.014,168.292,41.131,157.675
C02473=1033.222,-25.567,414.027,168.289,41.132,157.675
C02474=1033.215,-25.817,414.041,168.287,41.132,157.675
C02475=1033.210,-26.066,414.056,168.284,41.133,157.675
C02476=1033.203,-26.315,414.069,168.282,41.134,157.675
C02477=1033.197,-26.565,414.082,168.279,41.135,157.675
C02478=1033.191,-26.815,414.096,168.277,41.135,157.675
C02479=1033.185,-27.064,414.110,168.274,41.136,157.675
C02480=1033.179,-27.314,414.122,168.271,41.137,157.675
C02481=1033.172,-27.564,414.136,168.269,41.138,157.675
C02482=1033.166,-27.813,414.149,168.266,41.139,157.675
C02483=1033.160,-28.062,414.162,168.264,41.140,157.675
C02484=1033.153,-28.312,414.176,168.262,41.141,157.675
C02485=1033.147,-28.562,414.189,168.259,41.142,157.675
C02486=1033.141,-28.811,414.203,168.257,41.142,157.675
C02487=1033.134,-29.061,414.216,168.254,41.143,157.675
C02488=1033.128,-29.310,414.229,168.252,41.144,157.676
C02489=1033.122,-29.560,414.242,168.249,41.145,157.676
C02490=1033.115,-29.810,414.256,168.246,41.146,157.676
C02491=1033.109,-30.060,414.269,168.244,41.146,157.675
C02492=1033.103,-30.309,414.283,168.241,41.147,157.676
C02493=1033.097,-30.558,414.296,168.239,41.148,157.676
C02494=1033.090,-30.808,414.310,168.237,41.149,157.676
C02495=1033.084,-31.058,414.322,168.234,41.150,157.676
C02496=1033.078,-31.307,414.335,168.232,41.150,157.676
C02497=1033.072,-31.556,414.349,168.229,41.151,157.676
C02498=1033.065,-31.806,414.362,168.226,41.152,157.676
C02499=1033.059,-32.056,414.376,168.224,41.153,157.676
C02500=1033.053,-32.306,414.388,168.221,41.154,157.676
C02501=1033.047,-32.555,414.401,168.219,41.155,157.676
C02502=1033.040,-32.805,414.415,168.216,41.156,157.676
C02503=1033.034,-33.054,414.428,168.213,41.157,157.676
C02504=1033.028,-33.304,414.441,168.211,41.157,157.676
C02505=1033.021,-33.553,414.454,168.209,41.158,157.676
C02506=1033.015,-33.802,414.467,168.206,41.159,157.676
C02507=1033.008,-34.052,414.481,168.204,41.160,157.676
C02508=1033.003,-34.302,414.494,168.201,41.161,157.676
C02509=1032.996,-34.552,414.507,168.199,41.162,157.676
C02510=1032.990,-34.801,414.520,168.196,41.163,157.676
C02511=1032.984,-35.051,414.533,168.193,41.163,157.676
C02512=1032.978,-35.300,414.546,168.191,41.164,157.676
C02513=1032.971,-35.550,414.560,168.188,41.165,157.676
C02514=1032.964,-35.831,414.574,168.185,41.166,157.676
C02515=1032.957,-36.111,414.588,168.182,41.167,157.676
C02516=1032.951,-36.393,414.604,168.180,41.168,157.676
C02517=1032.944,-36.673,414.618,168.177,41.168,157.676
C02518=1032.937,-36.923,414.631,168.174,41.169,157.676
C02519=1032.931,-37.172,414.644,168.172,41.170,157.676
C02520=1032.925,-37.422,414.657,168.169,41.171,157.676
C02521=1032.919,-37.672,414.670,168.167,41.172,157.676
C02522=1032.913,-37.921,414.683,168.164,41.173,157.676
C02523=1032.907,-38.171,414.696,168.161,41.174,157.676
C02524=1032.900,-38.420,414.709,168.159,41.175,157.676
C02525=1032.895,-38.670,414.722,168.156,41.176,157.676
C02526=1032.888,-38.919,414.735,168.153,41.176,157.676
C02527=1032.882,-39.169,414.747,168.151,41.177,157.676
C02528=1032.875,-39.419,414.761,168.149,41.178,157.676
C02529=1032.869,-39.669,414.773,168.146,41.179,157.676
C02530=1032.863,-39.918,414.787,168.144,41.180,157.676
C02531=1032.856,-40.167,414.799,168.141,41.181,157.676
C02532=1032.850,-40.417,414.811,168.138,41.182,157.676
C02533=1032.844,-40.667,414.824,168.136,41.183,157.676
C02534=1032.838,-40.916,414.837,168.133,41.184,157.676
C02535=1032.831,-41.165,414.850,168.130,41.185,157.676
C02536=1032.825,-41.415,414.862,168.128,41.186,157.676
C02537=1032.819,-41.665,414.875,168.126,41.187,157.676
C02538=1032.812,-41.915,414.888,168.123,41.188,157.676
C02539=1032.806,-42.165,414.900,168.120,41.189,157.676
C02540=1032.800,-42.414,414.914,168.118,41.189,157.676
C02541=1032.794,-42.664,414.926,168.115,41.190,157.676
C02542=1032.788,-42.914,414.939,168.112,41.191,157.676
C02543=1032.781,-43.163,414.951,168.110,41.192,157.677
C02544=1032.775,-43.413,414.964,168.107,41.193,157.677
C02545=1032.769,-43.662,414.977,168.104,41.194,157.677
C02546=1032.762,-43.911,414.989,168.102,41.195,157.677
C02547=1032.756,-44.161,415.002,168.100,41.196,157.677
C02548=1032.750,-44.411,415.014,168.097,41.197,157.677
C02549=1032.744,-44.660,415.028,168.094,41.198,157.677
C02550=1032.737,-44.910,415.040,168.092,41.199,157.677
C02551=1032.732,-45.160,415.052,168.089,41.200,157.677
C02552=1032.725,-45.409,415.065,168.086,41.201,157.677
C02553=1032.719,-45.659,415.077,168.083,41.202,157.677
C02554=1032.713,-45.909,415.090,168.081,41.202,157.677
C02555=1032.707,-46.158,415.102,168.079,41.203,157.677
C02556=1032.700,-46.407,415.115,168.076,41.204,157.677
C02557=1032.694,-46.657,415.128,168.074,41.205,157.677
C02558=1032.688,-46.907,415.140,168.071,41.206,157.677
C02559=1032.682,-47.157,415.153,168.068,41.207,157.677
C02560=1032.676,-47.405,415.165,168.065,41.208,157.677
C02561=1032.670,-47.655,415.178,168.063,41.209,157.677
C02562=1032.664,-47.905,415.190,168.060,41.210,157.677
C02563=1032.657,-48.155,415.202,168.058,41.211,157.677
C02564=1032.651,-48.405,415.215,168.056,41.212,157.677
C02565=1032.645,-48.654,415.228,168.053,41.212,157.677
C02566=1032.639,-48.903,415.240,168.050,41.214,157.677
C02567=1032.633,-49.153,415.252,168.047,41.215,157.677
C02568=1032.627,-49.403,415.265,168.045,41.215,157.677
C02569=1032.620,-49.653,415.277,168.042,41.216,157.677
C02570=1032.614,-49.903,415.290,168.039,41.218,157.677
C02571=1032.608,-50.153,415.302,168.037,41.218,157.677
C02572=1032.602,-50.401,415.314,168.034,41.219,157.677
C02573=1032.596,-50.651,415.327,168.032,41.220,157.677
C02574=1032.589,-50.900,415.339,168.029,41.221,157.677
C02575=1032.583,-51.150,415.351,168.026,41.223,157.677
C02576=1032.577,-51.400,415.363,168.024,41.223,157.677
C02577=1032.570,-51.650,415.375,168.021,41.224,157.678
C02578=1032.563,-51.931,415.389,168.018,41.226,157.678
C02579=1032.557,-52.213,415.402,168.015,41.227,157.678
C02580=1032.549,-52.494,415.416,168.012,41.228,157.678
C02581=1032.542,-52.775,415.430,168.009,41.230,157.678
C02582=1032.535,-53.025,415.442,168.006,41.231,157.678
C02583=1032.530,-53.275,415.454,168.004,41.232,157.678
C02584=1032.523,-53.524,415.466,168.001,41.233,157.678
C02585=1032.516,-53.774,415.478,167.998,41.234,157.678
C02586=1032.510,-54.023,415.490,167.995,41.235,157.678
C02587=1032.504,-54.272,415.502,167.993,41.237,157.678
C02588=1032.498,-54.522,415.514,167.991,41.238,157.678
C02589=1032.491,-54.772,415.525,167.988,41.239,157.678
C02590=1032.485,-55.022,415.538,167.985,41.240,157.678
C02591=1032.479,-55.272,415.550,167.982,41.241,157.678
C02592=1032.472,-55.521,415.562,167.979,41.242,157.678
C02593=1032.467,-55.770,415.574,167.977,41.243,157.678
C02594=1032.460,-56.020,415.586,167.975,41.244,157.679
C02595=1032.454,-56.270,415.598,167.972,41.245,157.679
C02596=1032.447,-56.520,415.609,167.969,41.246,157.679
C02597=1032.441,-56.770,415.622,167.966,41.248,157.679
C02598=1032.435,-57.018,415.633,167.963,41.249,157.679
C02599=1032.429,-57.268,415.645,167.961,41.249,157.679
C02600=1032.423,-57.518,415.658,167.959,41.251,157.679
C02601=1032.416,-57.768,415.669,167.956,41.252,157.679
C02602=1032.410,-58.017,415.681,167.953,41.253,157.679
C02603=1032.404,-58.267,415.693,167.950,41.254,157.679
C02604=1032.398,-58.516,415.705,167.947,41.255,157.679
C02605=1032.391,-58.767,415.716,167.945,41.256,157.679
C02606=1032.385,-59.016,415.728,167.943,41.258,157.679
C02607=1032.379,-59.265,415.740,167.940,41.259,157.679
C02608=1032.373,-59.515,415.753,167.937,41.260,157.679
C02609=1032.366,-59.765,415.764,167.934,41.261,157.679
C02610=1032.360,-60.014,415.775,167.931,41.262,157.679
C02611=1032.355,-60.264,415.788,167.929,41.263,157.679
C02612=1032.348,-60.514,415.799,167.926,41.264,157.679
C02613=1032.342,-60.764,415.811,167.924,41.266,157.679
C02614=1032.335,-61.013,415.823,167.921,41.267,157.680
C02615=1032.330,-61.263,415.835,167.918,41.268,157.680
C02616=1032.323,-61.513,415.847,167.916,41.269,157.680
C02617=1032.317,-61.761,415.858,167.913,41.270,157.680
C02618=1032.311,-62.012,415.869,167.910,41.271,157.680
C02619=1032.305,-62.262,415.882,167.907,41.272,157.680
C02620=1032.299,-62.510,415.894,167.905,41.273,157.680
C02621=1032.293,-62.761,415.905,167.902,41.274,157.680
C02622=1032.286,-63.010,415.917,167.900,41.275,157.680
C02623=1032.281,-63.260,415.928,167.897,41.276,157.680
C02624=1032.274,-63.510,415.940,167.894,41.277,157.680
C02625=1032.268,-63.759,415.952,167.891,41.278,157.680
C02626=1032.262,-64.009,415.963,167.888,41.280,157.680
C02627=1032.255,-64.258,415.975,167.886,41.281,157.680
C02628=1032.250,-64.508,415.986,167.883,41.282,157.680
C02629=1032.244,-64.758,415.998,167.881,41.283,157.680
C02630=1032.237,-65.008,416.010,167.878,41.284,157.680
C02631=1032.231,-65.257,416.021,167.875,41.285,157.680
C02632=1032.225,-65.507,416.034,167.872,41.286,157.680
C02633=1032.220,-65.756,416.045,167.869,41.287,157.680
C02634=1032.213,-66.006,416.057,167.867,41.289,157.680
C02635=1032.207,-66.256,416.068,167.865,41.290,157.681
C02636=1032.201,-66.505,416.079,167.862,41.291,157.681
C02637=1032.195,-66.755,416.091,167.859,41.292,157.681
C02638=1032.189,-67.005,416.102,167.856,41.293,157.681
C02639=1032.183,-67.254,416.114,167.853,41.294,157.681
C02640=1032.177,-67.504,416.125,167.850,41.296,157.681
C02641=1032.170,-67.753,416.137,167.849,41.297,157.681
C02642=1032.161,-68.148,416.155,167.844,41.298,157.681
C02643=1032.151,-68.542,416.174,167.840,41.300,157.681
C02644=1032.142,-68.937,416.191,167.835,41.302,157.681
C02645=1032.133,-69.331,416.210,167.831,41.304,157.681
C02646=1032.124,-69.719,416.228,167.827,41.306,157.681
C02647=1032.114,-70.106,416.245,167.823,41.307,157.681
C02648=1032.105,-70.494,416.263,167.818,41.309,157.681
C02649=1032.095,-70.881,416.281,167.814,41.310,157.681
C02650=1032.089,-71.130,416.292,167.811,41.312,157.681
C02651=1032.083,-71.381,416.304,167.808,41.313,157.681
C02652=1032.077,-71.630,416.315,167.806,41.314,157.681
C02653=1032.071,-71.880,416.326,167.803,41.315,157.682
C02654=1032.066,-72.129,416.338,167.801,41.316,157.682
C02655=1032.059,-72.380,416.349,167.798,41.317,157.682
C02656=1032.054,-72.629,416.360,167.795,41.318,157.682
C02657=1032.047,-72.879,416.372,167.792,41.319,157.682
C02658=1032.041,-73.128,416.383,167.789,41.320,157.682
C02659=1032.035,-73.378,416.394,167.787,41.321,157.682
C02660=1032.030,-73.628,416.406,167.784,41.323,157.682
C02661=1032.024,-73.877,416.417,167.782,41.324,157.682
C02662=1032.017,-74.127,416.428,167.779,41.325,157.682
C02663=1032.012,-74.377,416.439,167.776,41.326,157.682
C02664=1032.006,-74.626,416.450,167.774,41.328,157.682
C02665=1032.000,-74.876,416.461,167.771,41.329,157.682
C02666=1031.994,-75.126,416.472,167.768,41.330,157.682
C02667=1031.987,-75.375,416.484,167.765,41.332,157.682
C02668=1031.981,-75.625,416.495,167.762,41.333,157.682
C02669=1031.974,-75.875,416.506,167.759,41.334,157.682
C02670=1031.969,-76.124,416.517,167.757,41.335,157.683
C02671=1031.963,-76.374,416.528,167.754,41.336,157.683
C02672=1031.957,-76.624,416.539,167.751,41.337,157.683
C02673=1031.951,-76.873,416.550,167.749,41.339,157.683
C02674=1031.945,-77.124,416.561,167.746,41.340,157.683
C02675=1031.938,-77.373,416.571,167.743,41.341,157.683
C02676=1031.932,-77.622,416.582,167.741,41.343,157.683
C02677=1031.926,-77.873,416.593,167.738,41.344,157.683
C02678=1031.920,-78.122,416.604,167.735,41.345,157.683
C02679=1031.914,-78.371,416.615,167.732,41.347,157.683
C02680=1031.908,-78.622,416.626,167.729,41.348,157.683
C02681=1031.902,-78.871,416.637,167.726,41.349,157.683
C02682=1031.897,-79.121,416.648,167.724,41.350,157.683
C02683=1031.890,-79.371,416.659,167.721,41.351,157.683
C02684=1031.884,-79.620,416.670,167.718,41.353,157.683
C02685=1031.878,-79.870,416.680,167.715,41.354,157.684
C02686=1031.872,-80.120,416.692,167.712,41.355,157.684
C02687=1031.866,-80.369,416.703,167.710,41.357,157.684
C02688=1031.860,-80.618,416.713,167.708,41.358,157.684
C02689=1031.853,-80.869,416.724,167.705,41.360,157.684
C02690=1031.847,-81.118,416.734,167.702,41.361,157.684
C02691=1031.841,-81.367,416.745,167.699,41.362,157.684
C02692=1031.835,-81.618,416.756,167.696,41.363,157.684
C02693=1031.828,-81.867,416.766,167.694,41.365,157.684
C02694=1031.823,-82.117,416.777,167.691,41.366,157.684
C02695=1031.816,-82.367,416.788,167.688,41.368,157.684
C02696=1031.810,-82.616,416.799,167.685,41.369,157.684
C02697=1031.804,-82.866,416.809,167.683,41.371,157.685
C02698=1031.798,-83.115,416.819,167.680,41.372,157.685
C02699=1031.792,-83.366,416.830,167.677,41.373,157.685
C02700=1031.786,-83.615,416.841,167.674,41.374,157.685
C02701=1031.779,-83.864,416.851,167.671,41.376,157.685
C02702=1031.773,-84.149,416.863,167.668,41.378,157.685
C02703=1031.765,-84.434,416.876,167.665,41.379,157.685
C02704=1031.759,-84.719,416.888,167.661,41.381,157.685
C02705=1031.752,-85.003,416.899,167.658,41.383,157.685
C02706=1031.745,-85.253,416.910,167.655,41.384,157.685
C02707=1031.739,-85.503,416.921,167.653,41.385,157.685
C02708=1031.734,-85.753,416.931,167.650,41.387,157.686
C02709=1031.727,-86.002,416.941,167.647,41.388,157.686
C02710=1031.721,-86.252,416.952,167.644,41.390,157.686
C02711=1031.715,-86.501,416.962,167.641,41.391,157.686
C02712=1031.709,-86.752,416.973,167.639,41.393,157.686
C02713=1031.703,-87.001,416.984,167.636,41.394,157.686
C02714=1031.697,-87.251,416.994,167.633,41.395,157.686
C02715=1031.691,-87.500,417.004,167.630,41.396,157.686
C02716=1031.685,-87.750,417.015,167.628,41.398,157.686
C02717=1031.679,-88.000,417.025,167.625,41.399,157.686
C02718=1031.672,-88.250,417.036,167.622,41.401,157.686
C02719=1031.667,-88.500,417.046,167.619,41.402,157.686
C02720=1031.661,-88.749,417.057,167.616,41.404,157.687
C02721=1031.655,-88.998,417.067,167.613,41.405,157.687
C02722=1031.649,-89.248,417.077,167.611,41.406,157.687
C02723=1031.643,-89.498,417.087,167.608,41.408,157.687
C02724=1031.637,-89.748,417.098,167.605,41.409,157.687
C02725=1031.630,-89.998,417.108,167.602,41.411,157.687
C02726=1031.625,-90.247,417.119,167.600,41.412,157.687
C02727=1031.618,-90.497,417.129,167.597,41.414,157.687
C02728=1031.613,-90.746,417.139,167.594,41.415,157.687
C02729=1031.607,-90.997,417.150,167.591,41.417,157.687
C02730=1031.601,-91.246,417.160,167.588,41.418,157.687
C02731=1031.595,-91.496,417.170,167.586,41.419,157.688
C02732=1031.589,-91.745,417.180,167.583,41.420,157.688
C02733=1031.583,-91.995,417.190,167.580,41.422,157.688
C02734=1031.577,-92.244,417.201,167.577,41.423,157.688
C02735=1031.571,-92.495,417.211,167.574,41.425,157.688
C02736=1031.564,-92.744,417.222,167.572,41.427,157.688
C02737=1031.559,-92.994,417.232,167.569,41.428,157.688
C02738=1031.553,-93.244,417.241,167.566,41.429,157.688
C02739=1031.547,-93.494,417.252,167.563,41.430,157.688
C02740=1031.541,-93.743,417.262,167.560,41.432,157.688
C02741=1031.535,-93.993,417.273,167.558,41.433,157.688
C02742=1031.530,-94.243,417.283,167.555,41.435,157.688
C02743=1031.523,-94.492,417.293,167.552,41.436,157.688
C02744=1031.518,-94.742,417.303,167.549,41.438,157.689
C02745=1031.512,-94.992,417.313,167.546,41.439,157.689
C02746=1031.506,-95.242,417.324,167.544,41.440,157.689
C02747=1031.500,-95.491,417.333,167.541,41.442,157.689
C02748=1031.494,-95.741,417.344,167.538,41.443,157.689
C02749=1031.488,-95.991,417.354,167.535,41.445,157.689
C02750=1031.482,-96.241,417.364,167.532,41.446,157.689
C02751=1031.476,-96.490,417.374,167.530,41.448,157.689
C02752=1031.470,-96.740,417.384,167.527,41.449,157.689
C02753=1031.464,-96.990,417.394,167.524,41.450,157.689
C02754=1031.459,-97.239,417.405,167.521,41.452,157.689
C02755=1031.452,-97.489,417.414,167.519,41.453,157.690
C02756=1031.447,-97.739,417.424,167.516,41.455,157.690
C02757=1031.441,-97.989,417.434,167.513,41.456,157.690
C02758=1031.434,-98.238,417.444,167.510,41.458,157.690
C02759=1031.429,-98.487,417.454,167.508,41.459,157.690
C02760=1031.423,-98.737,417.464,167.505,41.461,157.690
C02761=1031.417,-98.987,417.473,167.501,41.462,157.690
C02762=1031.411,-99.237,417.483,167.498,41.464,157.690
C02763=1031.405,-99.487,417.492,167.495,41.466,157.690
C02764=1031.399,-99.736,417.503,167.493,41.468,157.691
C02765=1031.393,-99.986,417.513,167.490,41.469,157.691
C02766=1031.386,-100.273,417.524,167.487,41.470,157.691
C02767=1031.379,-100.560,417.535,167.483,41.472,157.691
C02768=1031.372,-100.848,417.547,167.481,41.474,157.691
C02769=1031.366,-101.134,417.558,167.477,41.476,157.691
C02770=1031.359,-101.384,417.567,167.474,41.478,157.691
C02771=1031.353,-101.634,417.577,167.472,41.479,157.691
C02772=1031.347,-101.883,417.587,167.469,41.481,157.691
C02773=1031.341,-102.133,417.597,167.466,41.482,157.692
C02774=1031.336,-102.382,417.606,167.463,41.484,157.692
C02775=1031.330,-102.632,417.616,167.460,41.485,157.692
C02776=1031.323,-102.882,417.626,167.458,41.487,157.692
C02777=1031.318,-103.132,417.636,167.454,41.488,157.692
C02778=1031.312,-103.382,417.645,167.451,41.490,157.692
C02779=1031.306,-103.632,417.655,167.448,41.492,157.692
C02780=1031.299,-103.881,417.664,167.446,41.494,157.692
C02781=1031.294,-104.131,417.674,167.443,41.495,157.692
C02782=1031.288,-104.381,417.684,167.440,41.496,157.692
C02783=1031.282,-104.630,417.693,167.437,41.498,157.693
C02784=1031.276,-104.880,417.703,167.435,41.500,157.693
C02785=1031.270,-105.130,417.712,167.432,41.502,157.693
C02786=1031.264,-105.379,417.722,167.429,41.503,157.693
C02787=1031.259,-105.629,417.732,167.426,41.504,157.693
C02788=1031.253,-105.879,417.741,167.424,41.506,157.693
C02789=1031.247,-106.129,417.751,167.421,41.508,157.693
C02790=1031.240,-106.379,417.761,167.417,41.510,157.693
C02791=1031.235,-106.628,417.770,167.414,41.511,157.693
C02792=1031.229,-106.878,417.779,167.412,41.512,157.694
C02793=1031.224,-107.128,417.789,167.409,41.514,157.694
C02794=1031.217,-107.378,417.798,167.406,41.516,157.694
C02795=1031.211,-107.628,417.808,167.403,41.518,157.694
C02796=1031.206,-107.877,417.817,167.401,41.519,157.694
C02797=1031.199,-108.127,417.827,167.398,41.520,157.694
C02798=1031.193,-108.377,417.836,167.395,41.522,157.694
C02799=1031.187,-108.627,417.845,167.392,41.524,157.694
C02800=1031.182,-108.876,417.854,167.389,41.526,157.695
C02801=1031.176,-109.126,417.864,167.386,41.528,157.695
C02802=1031.169,-109.376,417.873,167.383,41.529,157.695
C02803=1031.163,-109.625,417.883,167.381,41.531,157.695
C02804=1031.158,-109.875,417.891,167.378,41.533,157.695
C02805=1031.152,-110.125,417.901,167.375,41.535,157.695
C02806=1031.146,-110.375,417.911,167.372,41.536,157.695
C02807=1031.140,-110.624,417.920,167.369,41.537,157.695
C02808=1031.134,-110.874,417.929,167.367,41.539,157.696
C02809=1031.128,-111.124,417.938,167.363,41.541,157.696
C02810=1031.122,-111.374,417.948,167.360,41.543,157.696
C02811=1031.117,-111.624,417.956,167.358,41.544,157.696
C02812=1031.110,-111.873,417.966,167.355,41.546,157.696
C02813=1031.104,-112.123,417.975,167.352,41.548,157.696
C02814=1031.099,-112.372,417.985,167.349,41.550,157.696
C02815=1031.093,-112.623,417.993,167.347,41.551,157.696
C02816=1031.087,-112.872,418.003,167.344,41.553,157.697
C02817=1031.081,-113.122,418.012,167.340,41.555,157.697
C02818=1031.075,-113.372,418.021,167.338,41.557,157.697
C02819=1031.070,-113.621,418.030,167.335,41.558,157.697
C02820=1031.064,-113.871,418.040,167.332,41.559,157.697
C02821=1031.058,-114.121,418.049,167.329,41.561,157.697
C02822=1031.052,-114.370,418.058,167.327,41.563,157.697
C02823=1031.046,-114.621,418.067,167.324,41.565,157.697
C02824=1031.040,-114.871,418.076,167.321,41.566,157.698
C02825=1031.034,-115.120,418.084,167.317,41.568,157.698
C02826=1031.028,-115.370,418.094,167.315,41.570,157.698
C02827=1031.022,-115.619,418.103,167.312,41.572,157.698
C02828=1031.016,-115.869,418.112,167.309,41.574,157.698
C02829=1031.010,-116.119,418.121,167.306,41.575,157.698
C02830=1031.004,-116.405,418.131,167.303,41.578,157.698
C02831=1030.997,-116.692,418.141,167.300,41.580,157.699
C02832=1030.990,-116.979,418.152,167.296,41.581,157.699
C02833=1030.983,-117.264,418.162,167.293,41.584,157.699
C02834=1030.978,-117.515,418.171,167.290,41.586,157.699
C02835=1030.972,-117.764,418.180,167.287,41.587,157.699
C02836=1030.966,-118.014,418.189,167.285,41.589,157.699
C02837=1030.960,-118.265,418.198,167.282,41.591,157.699
C02838=1030.954,-118.513,418.207,167.279,41.593,157.700
C02839=1030.948,-118.764,418.215,167.277,41.594,157.700
C02840=1030.943,-119.013,418.225,167.273,41.596,157.700
C02841=1030.937,-119.263,418.233,167.270,41.598,157.700
C02842=1030.931,-119.513,418.242,167.267,41.600,157.700
C02843=1030.924,-119.762,418.251,167.265,41.602,157.700
C02844=1030.919,-120.012,418.259,167.262,41.603,157.700
C02845=1030.913,-120.262,418.269,167.259,41.605,157.700
C02846=1030.908,-120.512,418.277,167.257,41.607,157.701
C02847=1030.901,-120.762,418.286,167.253,41.609,157.701
C02848=1030.896,-121.011,418.295,167.250,41.610,157.701
C02849=1030.890,-121.261,418.304,167.247,41.612,157.701
C02850=1030.884,-121.511,418.312,167.245,41.615,157.701
C02851=1030.878,-121.761,418.322,167.242,41.616,157.701
C02852=1030.872,-122.010,418.330,167.239,41.618,157.702
C02853=1030.866,-122.261,418.339,167.236,41.620,157.702
C02854=1030.861,-122.510,418.348,167.233,41.622,157.702
C02855=1030.854,-122.760,418.356,167.230,41.623,157.702
C02856=1030.849,-123.010,418.365,167.228,41.625,157.702
C02857=1030.843,-123.260,418.373,167.225,41.627,157.702
C02858=1030.838,-123.509,418.383,167.222,41.629,157.702
C02859=1030.832,-123.758,418.390,167.218,41.631,157.702
C02860=1030.826,-124.009,418.399,167.216,41.633,157.703
C02861=1030.820,-124.259,418.408,167.213,41.635,157.703
C02862=1030.814,-124.508,418.417,167.210,41.637,157.703
C02863=1030.808,-124.758,418.425,167.208,41.638,157.703
C02864=1030.802,-125.008,418.434,167.205,41.640,157.703
C02865=1030.796,-125.258,418.442,167.201,41.642,157.703
C02866=1030.791,-125.507,418.450,167.199,41.644,157.704
C02867=1030.785,-125.758,418.459,167.196,41.646,157.704
C02868=1030.779,-126.006,418.468,167.193,41.648,157.704
C02869=1030.773,-126.257,418.477,167.191,41.650,157.704
C02870=1030.767,-126.506,418.485,167.188,41.651,157.704
C02871=1030.762,-126.756,418.493,167.184,41.654,157.704
C02872=1030.756,-127.006,418.502,167.182,41.656,157.704
C02873=1030.750,-127.256,418.510,167.179,41.657,157.705
C02874=1030.745,-127.506,418.518,167.176,41.659,157.705
C02875=1030.738,-127.754,418.527,167.173,41.661,157.705
C02876=1030.733,-128.005,418.536,167.170,41.663,157.705
C02877=1030.728,-128.255,418.545,167.168,41.664,157.705
C02878=1030.724,-128.503,418.554,167.165,41.665,157.705
C02879=1030.720,-128.753,418.565,167.162,41.665,157.705
C02880=1030.717,-129.004,418.576,167.160,41.665,157.705
C02881=1030.715,-129.253,418.588,167.158,41.665,157.705
C02882=1030.712,-129.503,418.600,167.155,41.664,157.704
C02883=1030.712,-129.753,418.612,167.153,41.662,157.704
C02884=1030.711,-130.003,418.625,167.151,41.660,157.703
C02885=1030.711,-130.252,418.640,167.148,41.658,157.703
C02886=1030.712,-130.502,418.654,167.147,41.655,157.702
C02887=1030.714,-130.753,418.669,167.145,41.652,157.702
C02888=1030.715,-131.002,418.684,167.144,41.648,157.701
C02889=1030.718,-131.252,418.701,167.142,41.644,157.700
C02890=1030.721,-131.502,418.718,167.141,41.639,157.699
C02891=1030.725,-131.753,418.735,167.139,41.633,157.698
C02892=1030.730,-132.002,418.753,167.138,41.628,157.697
C02893=1030.735,-132.252,418.772,167.137,41.622,157.696
C02894=1030.415,-132.276,418.471,167.087,41.860,157.733
C02895=1030.409,-132.027,418.452,167.089,41.866,157.734
C02896=1030.405,-131.777,418.434,167.090,41.872,157.735
C02897=1030.401,-131.527,418.417,167.092,41.877,157.736
C02898=1030.398,-131.277,418.400,167.093,41.882,157.737
C02899=1030.394,-131.027,418.384,167.095,41.886,157.738
C02900=1030.392,-130.777,418.368,167.097,41.890,157.739
C02901=1030.392,-130.528,418.353,167.098,41.894,157.739
C02902=1030.390,-130.277,418.338,167.101,41.897,157.740
C02903=1030.390,-130.027,418.325,167.102,41.899,157.740
C02904=1030.391,-129.778,418.311,167.104,41.901,157.741
C02905=1030.392,-129.528,418.298,167.106,41.902,157.741
C02906=1030.393,-129.278,418.286,167.109,41.904,157.742
C02907=1030.396,-129.028,418.275,167.111,41.904,157.742
C02908=1030.399,-128.778,418.264,167.113,41.904,157.742
C02909=1030.403,-128.529,418.254,167.116,41.904,157.742
C02910=1030.407,-128.279,418.244,167.119,41.903,157.742
C02911=1030.412,-128.030,418.234,167.122,41.902,157.742
C02912=1030.418,-127.780,418.226,167.125,41.900,157.742
C02913=1030.423,-127.530,418.217,167.127,41.898,157.742
C02914=1030.429,-127.281,418.209,167.130,41.896,157.742
C02915=1030.434,-127.031,418.201,167.133,41.894,157.741
C02916=1030.440,-126.781,418.192,167.135,41.892,157.741
C02917=1030.447,-126.532,418.184,167.139,41.890,157.741
C02918=1030.452,-126.282,418.175,167.142,41.888,157.741
C02919=1030.458,-126.032,418.167,167.144,41.886,157.741
C02920=1030.464,-125.783,418.158,167.147,41.884,157.741
C02921=1030.470,-125.532,418.149,167.151,41.883,157.741
C02922=1030.476,-125.283,418.142,167.153,41.880,157.740
C02923=1030.481,-125.032,418.133,167.156,41.878,157.740
C02924=1030.488,-124.784,418.124,167.159,41.877,157.740
C02925=1030.493,-124.534,418.116,167.161,41.875,157.740
C02926=1030.499,-124.283,418.107,167.165,41.872,157.740
C02927=1030.505,-124.034,418.099,167.168,41.870,157.740
C02928=1030.511,-123.784,418.090,167.170,41.869,157.739
C02929=1030.516,-123.535,418.081,167.173,41.867,157.739
C02930=1030.522,-123.285,418.072,167.176,41.865,157.739
C02931=1030.528,-123.035,418.064,167.178,41.863,157.739
C02932=1030.533,-122.785,418.056,167.182,41.861,157.739
C02933=1030.540,-122.535,418.046,167.185,41.859,157.739
C02934=1030.545,-122.285,418.038,167.187,41.857,157.739
C02935=1030.551,-122.035,418.029,167.190,41.855,157.738
C02936=1030.557,-121.786,418.021,167.193,41.854,157.738
C02937=1030.563,-121.536,418.011,167.197,41.852,157.738
C02938=1030.568,-121.286,418.003,167.199,41.850,157.738
C02939=1030.575,-121.036,417.994,167.202,41.848,157.738
C02940=1030.580,-120.787,417.985,167.205,41.846,157.738
C02941=1030.586,-120.537,417.976,167.207,41.844,157.738
C02942=1030.591,-120.287,417.968,167.210,41.842,157.737
C02943=1030.598,-120.038,417.959,167.214,41.840,157.737
C02944=1030.604,-119.788,417.950,167.216,41.839,157.737
C02945=1030.609,-119.537,417.942,167.219,41.837,157.737
C02946=1030.615,-119.288,417.932,167.222,41.835,157.737
C02947=1030.621,-119.038,417.924,167.224,41.833,157.737
C02948=1030.627,-118.789,417.915,167.228,41.831,157.737
C02949=1030.633,-118.538,417.906,167.231,41.829,157.737
C02950=1030.639,-118.289,417.897,167.233,41.827,157.736
C02951=1030.645,-118.039,417.888,167.236,41.825,157.736
C02952=1030.650,-117.789,417.880,167.239,41.824,157.736
C02953=1030.657,-117.540,417.871,167.242,41.822,157.736
C02954=1030.662,-117.290,417.862,167.245,41.820,157.736
C02955=1030.669,-117.003,417.851,167.248,41.818,157.736
C02956=1030.676,-116.717,417.841,167.252,41.816,157.736
C02957=1030.682,-116.431,417.831,167.255,41.814,157.735
C02958=1030.689,-116.144,417.820,167.258,41.812,157.735
C02959=1030.695,-115.895,417.812,167.261,41.810,157.735
C02960=1030.701,-115.645,417.803,167.263,41.808,157.735
C02961=1030.707,-115.395,417.793,167.267,41.806,157.735
C02962=1030.712,-115.145,417.785,167.270,41.804,157.735
C02963=1030.718,-114.895,417.775,167.272,41.802,157.735
C02964=1030.724,-114.646,417.767,167.275,41.801,157.734
C02965=1030.730,-114.396,417.757,167.278,41.799,157.734
C02966=1030.736,-114.146,417.748,167.281,41.797,157.734
C02967=1030.741,-113.896,417.739,167.284,41.795,157.734
C02968=1030.747,-113.647,417.730,167.287,41.793,157.734
C02969=1030.753,-113.396,417.721,167.290,41.792,157.734
C02970=1030.759,-113.147,417.712,167.292,41.790,157.734
C02971=1030.765,-112.897,417.702,167.295,41.788,157.734
C02972=1030.771,-112.647,417.693,167.298,41.786,157.733
C02973=1030.777,-112.398,417.685,167.301,41.785,157.733
C02974=1030.783,-112.148,417.675,167.304,41.783,157.733
C02975=1030.789,-111.899,417.666,167.307,41.781,157.733
C02976=1030.795,-111.649,417.657,167.310,41.780,157.733
C02977=1030.801,-111.399,417.647,167.313,41.778,157.733
C02978=1030.806,-111.149,417.639,167.315,41.776,157.733
C02979=1030.812,-110.900,417.629,167.318,41.775,157.733
C02980=1030.819,-110.650,417.620,167.321,41.773,157.732
C02981=1030.825,-110.400,417.610,167.324,41.771,157.732
C02982=1030.830,-110.150,417.602,167.327,41.769,157.732
C02983=1030.836,-109.900,417.592,167.330,41.768,157.732
C02984=1030.842,-109.651,417.583,167.333,41.766,157.732
C02985=1030.848,-109.402,417.573,167.335,41.764,157.732
C02986=1030.854,-109.151,417.564,167.338,41.762,157.732
C02987=1030.860,-108.901,417.555,167.341,41.761,157.732
C02988=1030.865,-108.651,417.545,167.344,41.759,157.731
C02989=1030.871,-108.402,417.536,167.347,41.757,157.731
C02990=1030.877,-108.152,417.526,167.350,41.755,157.731
C02991=1030.883,-107.902,417.517,167.353,41.753,157.731
C02992=1030.889,-107.652,417.508,167.355,41.752,157.731
C02993=1030.895,-107.403,417.498,167.358,41.750,157.731
C02994=1030.901,-107.153,417.489,167.361,41.748,157.731
C02995=1030.907,-106.903,417.479,167.365,41.747,157.731
C02996=1030.913,-106.654,417.470,167.367,41.745,157.731
C02997=1030.919,-106.405,417.460,167.370,41.743,157.730
C02998=1030.925,-106.154,417.452,167.373,41.742,157.730
C02999=1030.930,-105.904,417.441,167.375,41.740,157.730
C03000=1030.936,-105.654,417.432,167.378,41.738,157.730
C03001=1030.943,-105.404,417.422,167.381,41.736,157.730
C03002=1030.948,-105.155,417.413,167.384,41.735,157.730
C03003=1030.954,-104.905,417.404,167.386,41.734,157.730
C03004=1030.960,-104.656,417.394,167.389,41.732,157.730
C03005=1030.966,-104.406,417.384,167.393,41.730,157.729
C03006=1030.972,-104.156,417.374,167.396,41.728,157.729
C03007=1030.978,-103.907,417.365,167.398,41.726,157.729
C03008=1030.984,-103.657,417.355,167.401,41.725,157.729
C03009=1030.990,-103.407,417.346,167.404,41.724,157.729
C03010=1030.995,-103.157,417.336,167.407,41.722,157.729
C03011=1031.002,-102.907,417.326,167.409,41.720,157.729
C03012=1031.008,-102.657,417.317,167.412,41.718,157.729
C03013=1031.014,-102.408,417.307,167.415,41.717,157.729
C03014=1031.019,-102.158,417.297,167.418,41.716,157.729
C03015=1031.025,-101.908,417.288,167.421,41.714,157.728
C03016=1031.031,-101.659,417.278,167.424,41.712,157.728
C03017=1031.038,-101.409,417.268,167.427,41.710,157.728
C03018=1031.043,-101.159,417.258,167.430,41.709,157.728
C03019=1031.050,-100.873,417.247,167.432,41.707,157.728
C03020=1031.057,-100.585,417.236,167.436,41.705,157.728
C03021=1031.064,-100.299,417.225,167.440,41.703,157.728
C03022=1031.071,-100.011,417.213,167.442,41.701,157.728
C03023=1031.076,-99.761,417.203,167.445,41.700,157.728
C03024=1031.082,-99.512,417.194,167.448,41.698,157.727
C03025=1031.088,-99.262,417.185,167.451,41.697,157.727
C03026=1031.095,-99.013,417.174,167.453,41.695,157.727
C03027=1031.100,-98.763,417.164,167.457,41.693,157.727
C03028=1031.106,-98.513,417.155,167.460,41.692,157.727
C03029=1031.112,-98.264,417.145,167.463,41.690,157.727
C03030=1031.119,-98.014,417.135,167.465,41.688,157.727
C03031=1031.124,-97.764,417.124,167.468,41.687,157.727
C03032=1031.131,-97.514,417.115,167.471,41.685,157.726
C03033=1031.137,-97.265,417.105,167.474,41.684,157.726
C03034=1031.142,-97.015,417.095,167.476,41.682,157.726
C03035=1031.149,-96.765,417.085,167.479,41.681,157.726
C03036=1031.154,-96.515,417.075,167.482,41.679,157.726
C03037=1031.160,-96.265,417.065,167.485,41.678,157.726
C03038=1031.166,-96.016,417.054,167.488,41.676,157.726
C03039=1031.172,-95.766,417.045,167.490,41.675,157.726
C03040=1031.178,-95.516,417.035,167.493,41.674,157.726
C03041=1031.183,-95.267,417.024,167.496,41.672,157.726
C03042=1031.189,-95.017,417.014,167.499,41.670,157.726
C03043=1031.195,-94.767,417.004,167.501,41.669,157.726
C03044=1031.201,-94.517,416.994,167.504,41.667,157.725
C03045=1031.207,-94.267,416.984,167.508,41.666,157.725
C03046=1031.213,-94.018,416.973,167.511,41.664,157.725
C03047=1031.219,-93.768,416.963,167.513,41.663,157.725
C03048=1031.225,-93.518,416.954,167.516,41.662,157.725
C03049=1031.231,-93.269,416.943,167.519,41.660,157.725
C03050=1031.237,-93.019,416.933,167.522,41.658,157.725
C03051=1031.243,-92.770,416.922,167.525,41.657,157.725
C03052=1031.249,-92.520,416.913,167.527,41.655,157.725
C03053=1031.254,-92.270,416.902,167.530,41.654,157.725
C03054=1031.261,-92.020,416.892,167.533,41.652,157.725
C03055=1031.266,-91.771,416.881,167.536,41.651,157.724
C03056=1031.273,-91.521,416.872,167.539,41.650,157.724
C03057=1031.278,-91.272,416.861,167.541,41.648,157.724
C03058=1031.284,-91.022,416.851,167.544,41.647,157.724
C03059=1031.290,-90.772,416.840,167.547,41.645,157.724
C03060=1031.296,-90.522,416.830,167.550,41.643,157.724
C03061=1031.303,-90.272,416.820,167.552,41.642,157.724
C03062=1031.308,-90.022,416.809,167.555,41.641,157.724
C03063=1031.315,-89.773,416.799,167.558,41.640,157.724
C03064=1031.320,-89.523,416.789,167.561,41.638,157.724
C03065=1031.327,-89.274,416.779,167.564,41.637,157.724
C03066=1031.332,-89.024,416.768,167.566,41.635,157.724
C03067=1031.338,-88.774,416.758,167.569,41.633,157.723
C03068=1031.344,-88.525,416.747,167.572,41.632,157.723
C03069=1031.350,-88.274,416.737,167.575,41.630,157.723
C03070=1031.357,-88.025,416.727,167.578,41.629,157.723
C03071=1031.362,-87.776,416.716,167.580,41.628,157.723
C03072=1031.369,-87.526,416.706,167.583,41.626,157.723
C03073=1031.374,-87.276,416.695,167.586,41.625,157.723
C03074=1031.380,-87.026,416.685,167.589,41.623,157.723
C03075=1031.387,-86.776,416.674,167.591,41.622,157.723
C03076=1031.393,-86.527,416.664,167.594,41.620,157.723
C03077=1031.399,-86.277,416.654,167.597,41.619,157.722
C03078=1031.405,-86.028,416.643,167.600,41.618,157.722
C03079=1031.411,-85.778,416.633,167.602,41.616,157.722
C03080=1031.417,-85.528,416.622,167.605,41.615,157.722
C03081=1031.423,-85.278,416.611,167.609,41.613,157.722
C03082=1031.429,-85.029,416.601,167.612,41.611,157.722
C03083=1031.436,-84.744,416.589,167.615,41.610,157.722
C03084=1031.443,-84.460,416.577,167.617,41.608,157.722
C03085=1031.450,-84.174,416.565,167.621,41.606,157.722
C03086=1031.457,-83.890,416.553,167.624,41.605,157.722
C03087=1031.463,-83.640,416.543,167.627,41.604,157.722
C03088=1031.469,-83.391,416.532,167.629,41.602,157.721
C03089=1031.475,-83.141,416.521,167.632,41.600,157.721
C03090=1031.481,-82.891,416.511,167.635,41.599,157.721
C03091=1031.487,-82.641,416.500,167.638,41.597,157.721
C03092=1031.494,-82.392,416.490,167.641,41.596,157.721
C03093=1031.500,-82.142,416.479,167.643,41.595,157.721
C03094=1031.506,-81.893,416.468,167.646,41.594,157.721
C03095=1031.512,-81.643,416.458,167.649,41.592,157.721
C03096=1031.518,-81.393,416.447,167.652,41.590,157.721
C03097=1031.525,-81.143,416.437,167.654,41.589,157.721
C03098=1031.531,-80.894,416.426,167.657,41.587,157.721
C03099=1031.537,-80.644,416.415,167.661,41.586,157.721
C03100=1031.543,-80.395,416.404,167.664,41.584,157.720
C03101=1031.549,-80.144,416.394,167.666,41.583,157.720
C03102=1031.555,-79.894,416.383,167.669,41.582,157.720
C03103=1031.561,-79.645,416.372,167.671,41.581,157.720
C03104=1031.567,-79.396,416.362,167.674,41.579,157.720
C03105=1031.573,-79.146,416.351,167.677,41.578,157.720
C03106=1031.579,-78.896,416.340,167.680,41.576,157.720
C03107=1031.585,-78.646,416.329,167.682,41.575,157.720
C03108=1031.591,-78.397,416.318,167.685,41.573,157.720
C03109=1031.597,-78.147,416.307,167.688,41.572,157.720
C03110=1031.603,-77.897,416.296,167.691,41.571,157.720
C03111=1031.609,-77.648,416.285,167.694,41.569,157.720
C03112=1031.616,-77.398,416.274,167.696,41.568,157.720
C03113=1031.622,-77.148,416.263,167.699,41.567,157.719
C03114=1031.628,-76.898,416.252,167.702,41.566,157.719
C03115=1031.634,-76.649,416.241,167.705,41.565,157.719
C03116=1031.640,-76.400,416.230,167.708,41.563,157.719
C03117=1031.646,-76.150,416.218,167.711,41.562,157.719
C03118=1031.652,-75.900,416.208,167.713,41.560,157.719
C03119=1031.657,-75.651,416.197,167.716,41.559,157.719
C03120=1031.665,-75.401,416.186,167.719,41.558,157.719
C03121=1031.670,-75.151,416.175,167.722,41.556,157.719
C03122=1031.677,-74.901,416.164,167.725,41.555,157.719
C03123=1031.682,-74.652,416.153,167.727,41.553,157.719
C03124=1031.689,-74.401,416.142,167.729,41.552,157.719
C03125=1031.695,-74.153,416.130,167.732,41.551,157.719
C03126=1031.700,-73.903,416.119,167.735,41.550,157.719
C03127=1031.707,-73.653,416.108,167.738,41.549,157.719
C03128=1031.713,-73.403,416.097,167.741,41.548,157.718
C03129=1031.718,-73.153,416.085,167.743,41.547,157.718
C03130=1031.724,-72.904,416.074,167.746,41.545,157.718
C03131=1031.730,-72.655,416.063,167.749,41.544,157.718
C03132=1031.736,-72.404,416.052,167.752,41.543,157.718
C03133=1031.742,-72.155,416.041,167.755,41.542,157.718
C03134=1031.749,-71.905,416.029,167.757,41.541,157.718
C03135=1031.754,-71.655,416.017,167.759,41.539,157.718
C03136=1031.760,-71.405,416.006,167.762,41.538,157.718
C03137=1031.766,-71.156,415.994,167.765,41.537,157.718
C03138=1031.772,-70.907,415.984,167.768,41.536,157.718
C03139=1031.778,-70.657,415.972,167.771,41.535,157.718
C03140=1031.784,-70.408,415.961,167.774,41.533,157.718
C03141=1031.790,-70.157,415.949,167.776,41.532,157.718
C03142=1031.796,-69.908,415.938,167.778,41.531,157.718
C03143=1031.802,-69.658,415.926,167.781,41.530,157.718
C03144=1031.808,-69.409,415.915,167.784,41.529,157.718
C03145=1031.815,-69.159,415.903,167.787,41.527,157.718
C03146=1031.820,-68.909,415.892,167.790,41.526,157.718
C03147=1031.827,-68.627,415.879,167.793,41.525,157.718
C03148=1031.834,-68.344,415.866,167.795,41.523,157.717
C03149=1031.841,-68.062,415.853,167.799,41.522,157.717
C03150=1031.847,-67.779,415.840,167.802,41.521,157.717
C03151=1031.854,-67.529,415.828,167.805,41.519,157.717
C03152=1031.859,-67.280,415.817,167.808,41.518,157.717
C03153=1031.866,-67.030,415.805,167.811,41.517,157.717
C03154=1031.871,-66.781,415.794,167.812,41.516,157.717
C03155=1031.878,-66.531,415.782,167.815,41.515,157.717
C03156=1031.884,-66.281,415.771,167.818,41.514,157.717
C03157=1031.889,-66.031,415.759,167.821,41.513,157.717
C03158=1031.896,-65.781,415.747,167.824,41.512,157.717
C03159=1031.902,-65.532,415.737,167.827,41.510,157.717
C03160=1031.908,-65.282,415.725,167.829,41.509,157.717
C03161=1031.914,-65.033,415.712,167.832,41.508,157.717
C03162=1031.920,-64.783,415.701,167.834,41.507,157.717
C03163=1031.927,-64.533,415.689,167.837,41.506,157.717
C03164=1031.932,-64.284,415.678,167.840,41.505,157.717
C03165=1031.939,-64.034,415.666,167.843,41.504,157.717
C03166=1031.945,-63.784,415.655,167.845,41.502,157.717
C03167=1031.951,-63.535,415.643,167.848,41.501,157.717
C03168=1031.957,-63.285,415.632,167.851,41.500,157.716
C03169=1031.963,-63.036,415.620,167.853,41.499,157.716
C03170=1031.969,-62.786,415.608,167.856,41.497,157.716
C03171=1031.975,-62.536,415.596,167.859,41.496,157.716
C03172=1031.981,-62.287,415.585,167.862,41.495,157.716
C03173=1031.988,-62.037,415.573,167.864,41.494,157.716
C03174=1031.994,-61.787,415.561,167.867,41.493,157.716
C03175=1032.000,-61.538,415.549,167.870,41.491,157.716
C03176=1032.006,-61.288,415.538,167.872,41.490,157.716
C03177=1032.013,-61.038,415.526,167.875,41.489,157.716
C03178=1032.018,-60.789,415.514,167.878,41.488,157.716
C03179=1032.024,-60.539,415.503,167.880,41.486,157.716
C03180=1032.031,-60.289,415.491,167.883,41.485,157.716
C03181=1032.038,-60.040,415.479,167.886,41.484,157.716
C03182=1032.043,-59.790,415.467,167.889,41.483,157.716
C03183=1032.049,-59.540,415.455,167.891,41.482,157.716
C03184=1032.056,-59.291,415.443,167.894,41.481,157.716
C03185=1032.062,-59.042,415.432,167.896,41.480,157.716
C03186=1032.067,-58.791,415.420,167.899,41.479,157.716
C03187=1032.074,-58.542,415.408,167.902,41.478,157.715
C03188=1032.081,-58.292,415.396,167.905,41.476,157.715
C03189=1032.087,-58.043,415.385,167.908,41.475,157.715
C03190=1032.092,-57.793,415.373,167.910,41.474,157.715
C03191=1032.099,-57.543,415.361,167.913,41.473,157.715
C03192=1032.106,-57.294,415.349,167.915,41.472,157.715
C03193=1032.112,-57.044,415.336,167.918,41.470,157.715
C03194=1032.117,-56.794,415.325,167.921,41.469,157.715
C03195=1032.124,-56.545,415.313,167.924,41.468,157.715
C03196=1032.131,-56.295,415.301,167.926,41.467,157.715
C03197=1032.137,-56.045,415.289,167.928,41.465,157.715
C03198=1032.143,-55.796,415.277,167.931,41.464,157.715
C03199=1032.149,-55.546,415.266,167.934,41.463,157.715
C03200=1032.155,-55.296,415.253,167.937,41.462,157.715
C03201=1032.162,-55.047,415.241,167.940,41.461,157.715
C03202=1032.168,-54.797,415.229,167.943,41.459,157.715
C03203=1032.177,-54.421,415.211,167.947,41.458,157.715
C03204=1032.187,-54.045,415.194,167.950,41.456,157.714
C03205=1032.197,-53.668,415.175,167.954,41.455,157.714
C03206=1032.205,-53.291,415.157,167.959,41.453,157.714
C03207=1032.216,-52.887,415.138,167.962,41.451,157.714
C03208=1032.227,-52.483,415.118,167.967,41.449,157.714
C03209=1032.237,-52.079,415.099,167.971,41.447,157.714
C03210=1032.247,-51.675,415.079,167.976,41.445,157.714
C03211=1032.253,-51.426,415.067,167.979,41.444,157.714
C03212=1032.259,-51.176,415.055,167.981,41.442,157.714
C03213=1032.266,-50.927,415.043,167.984,41.441,157.714
C03214=1032.273,-50.677,415.031,167.986,41.440,157.714
C03215=1032.278,-50.427,415.018,167.989,41.439,157.714
C03216=1032.284,-50.177,415.006,167.992,41.438,157.714
C03217=1032.291,-49.928,414.994,167.995,41.437,157.714
C03218=1032.297,-49.678,414.981,167.997,41.436,157.714
C03219=1032.303,-49.428,414.969,167.999,41.435,157.714
C03220=1032.309,-49.178,414.957,168.002,41.434,157.713
C03221=1032.315,-48.929,414.944,168.005,41.433,157.713
C03222=1032.321,-48.680,414.931,168.007,41.432,157.713
C03223=1032.328,-48.430,414.919,168.010,41.431,157.713
C03224=1032.334,-48.181,414.907,168.013,41.430,157.713
C03225=1032.339,-47.931,414.894,168.016,41.429,157.713
C03226=1032.346,-47.681,414.882,168.018,41.428,157.713
C03227=1032.352,-47.432,414.869,168.020,41.427,157.713
C03228=1032.358,-47.182,414.856,168.023,41.426,157.713
C03229=1032.364,-46.932,414.844,168.026,41.425,157.713
C03230=1032.371,-46.682,414.832,168.028,41.424,157.713
C03231=1032.377,-46.433,414.819,168.031,41.423,157.713
C03232=1032.383,-46.183,414.806,168.034,41.422,157.713
C03233=1032.390,-45.934,414.794,168.037,41.421,157.713
C03234=1032.395,-45.684,414.781,168.039,41.420,157.713
C03235=1032.401,-45.434,414.769,168.041,41.419,157.713
C03236=1032.408,-45.185,414.756,168.044,41.418,157.713
C03237=1032.414,-44.935,414.744,168.046,41.417,157.713
C03238=1032.420,-44.685,414.731,168.049,41.416,157.713
C03239=1032.427,-44.436,414.718,168.052,41.415,157.713
C03240=1032.433,-44.186,414.706,168.055,41.414,157.713
C03241=1032.439,-43.937,414.693,168.057,41.413,157.713
C03242=1032.445,-43.687,414.681,168.060,41.412,157.713
C03243=1032.452,-43.438,414.668,168.062,41.411,157.713
C03244=1032.458,-43.188,414.656,168.065,41.410,157.713
C03245=1032.464,-42.939,414.642,168.067,41.409,157.713
C03246=1032.471,-42.689,414.630,168.070,41.408,157.713
C03247=1032.476,-42.439,414.618,168.073,41.407,157.713
C03248=1032.483,-42.190,414.604,168.076,41.406,157.713
C03249=1032.489,-41.940,414.592,168.078,41.405,157.713
C03250=1032.495,-41.690,414.580,168.081,41.404,157.713
C03251=1032.501,-41.441,414.567,168.083,41.403,157.712
C03252=1032.507,-41.191,414.554,168.085,41.402,157.712
C03253=1032.514,-40.942,414.541,168.088,41.401,157.712
C03254=1032.520,-40.692,414.529,168.091,41.400,157.712
C03255=1032.526,-40.443,414.516,168.094,41.399,157.712
C03256=1032.532,-40.193,414.503,168.096,41.398,157.712
C03257=1032.539,-39.944,414.491,168.099,41.397,157.712
C03258=1032.546,-39.694,414.477,168.102,41.396,157.712
C03259=1032.552,-39.444,414.465,168.104,41.395,157.712
C03260=1032.558,-39.195,414.452,168.106,41.394,157.712
C03261=1032.565,-38.945,414.440,168.109,41.393,157.712
C03262=1032.571,-38.696,414.426,168.112,41.392,157.712
C03263=1032.577,-38.446,414.414,168.114,41.391,157.712
C03264=1032.583,-38.197,414.401,168.117,41.390,157.712
C03265=1032.589,-37.947,414.388,168.120,41.389,157.712
C03266=1032.595,-37.697,414.375,168.122,41.388,157.712
C03267=1032.601,-37.448,414.362,168.125,41.387,157.712
C03268=1032.608,-37.198,414.349,168.127,41.386,157.712
C03269=1032.614,-36.948,414.335,168.129,41.385,157.712
C03270=1032.620,-36.698,414.323,168.132,41.384,157.712
C03271=1032.626,-36.418,414.307,168.135,41.383,157.712
C03272=1032.634,-36.137,414.293,168.138,41.382,157.712
C03273=1032.641,-35.857,414.278,168.141,41.381,157.712
C03274=1032.648,-35.575,414.264,168.144,41.380,157.712
C03275=1032.654,-35.326,414.250,168.147,41.380,157.712
C03276=1032.660,-35.076,414.238,168.149,41.379,157.712
C03277=1032.666,-34.827,414.225,168.152,41.378,157.712
C03278=1032.673,-34.577,414.211,168.154,41.377,157.712
C03279=1032.678,-34.328,414.199,168.156,41.376,157.712
C03280=1032.685,-34.078,414.185,168.159,41.375,157.712
C03281=1032.691,-33.828,414.172,168.162,41.374,157.712
C03282=1032.697,-33.578,414.159,168.164,41.374,157.712
C03283=1032.704,-33.329,414.146,168.167,41.373,157.712
C03284=1032.710,-33.080,414.133,168.170,41.372,157.712
C03285=1032.716,-32.831,414.120,168.172,41.371,157.712
C03286=1032.723,-32.580,414.107,168.175,41.370,157.712
C03287=1032.729,-32.331,414.093,168.177,41.369,157.712
C03288=1032.735,-32.082,414.080,168.179,41.368,157.712
C03289=1032.741,-31.832,414.067,168.182,41.367,157.712
C03290=1032.748,-31.582,414.054,168.184,41.366,157.712
C03291=1032.754,-31.332,414.041,168.187,41.365,157.712
C03292=1032.760,-31.083,414.027,168.190,41.364,157.712
C03293=1032.766,-30.834,414.014,168.192,41.363,157.712
C03294=1032.773,-30.584,414.000,168.195,41.362,157.711
C03295=1032.778,-30.334,413.987,168.198,41.361,157.711
C03296=1032.785,-30.084,413.974,168.199,41.360,157.711
C03297=1032.791,-29.835,413.961,168.202,41.359,157.711
C03298=1032.798,-29.585,413.947,168.205,41.358,157.711
C03299=1032.804,-29.336,413.934,168.207,41.358,157.711
C03300=1032.810,-29.087,413.921,168.210,41.357,157.711
C03301=1032.816,-28.836,413.908,168.213,41.356,157.711
C03302=1032.823,-28.587,413.894,168.215,41.355,157.711
C03303=1032.829,-28.338,413.881,168.218,41.354,157.711
C03304=1032.835,-28.088,413.868,168.220,41.353,157.711
C03305=1032.842,-27.838,413.854,168.222,41.352,157.711
C03306=1032.848,-27.589,413.841,168.225,41.351,157.711
C03307=1032.854,-27.340,413.828,168.227,41.350,157.711
C03308=1032.861,-27.090,413.814,168.230,41.350,157.711
C03309=1032.867,-26.841,413.801,168.233,41.349,157.711
C03310=1032.873,-26.591,413.787,168.235,41.348,157.711
C03311=1032.880,-26.341,413.773,168.238,41.347,157.711
C03312=1032.886,-26.092,413.760,168.240,41.347,157.711
C03313=1032.891,-25.842,413.746,168.243,41.345,157.711
C03314=1032.898,-25.592,413.733,168.246,41.344,157.711
C03315=1032.904,-25.343,413.719,168.248,41.344,157.711
C03316=1032.911,-25.094,413.706,168.251,41.343,157.711
C03317=1032.917,-24.843,413.692,168.252,41.342,157.711
C03318=1032.923,-24.594,413.678,168.255,41.341,157.711
C03319=1032.929,-24.345,413.665,168.257,41.340,157.711
C03320=1032.935,-24.095,413.651,168.260,41.340,157.711
C03321=1032.941,-23.845,413.638,168.263,41.339,157.711
C03322=1032.948,-23.596,413.624,168.265,41.338,157.711
C03323=1032.954,-23.346,413.610,168.268,41.337,157.711
C03324=1032.960,-23.097,413.596,168.270,41.337,157.711
C03325=1032.966,-22.848,413.583,168.273,41.336,157.711
C03326=1032.973,-22.598,413.569,168.275,41.335,157.711
C03327=1032.979,-22.348,413.555,168.277,41.334,157.711
C03328=1032.986,-22.098,413.542,168.281,41.333,157.711
C03329=1032.992,-21.849,413.529,168.282,41.332,157.711
C03330=1032.997,-21.600,413.515,168.285,41.331,157.711
C03331=1033.004,-21.350,413.501,168.287,41.330,157.711
C03332=1033.011,-21.101,413.487,168.290,41.330,157.711
C03333=1033.017,-20.851,413.473,168.292,41.329,157.711
C03334=1033.023,-20.601,413.460,168.295,41.328,157.711
C03335=1033.030,-20.320,413.444,168.298,41.327,157.711
C03336=1033.037,-20.038,413.428,168.301,41.326,157.711
C03337=1033.044,-19.757,413.413,168.304,41.326,157.711
C03338=1033.051,-19.474,413.397,168.307,41.325,157.711
C03339=1033.058,-19.226,413.383,168.308,41.324,157.711
C03340=1033.064,-18.976,413.370,168.311,41.323,157.711
C03341=1033.070,-18.726,413.356,168.313,41.322,157.711
C03342=1033.076,-18.477,413.343,168.316,41.321,157.711
C03343=1033.083,-18.227,413.328,168.318,41.321,157.711
C03344=1033.089,-17.978,413.314,168.321,41.320,157.711
C03345=1033.096,-17.728,413.301,168.324,41.318,157.711
C03346=1033.101,-17.478,413.287,168.326,41.318,157.711
C03347=1033.108,-17.229,413.272,168.329,41.317,157.711
C03348=1033.114,-16.980,413.259,168.331,41.316,157.711
C03349=1033.120,-16.730,413.245,168.334,41.315,157.711
C03350=1033.127,-16.481,413.231,168.335,41.314,157.711
C03351=1033.134,-16.231,413.217,168.338,41.313,157.711
C03352=1033.139,-15.981,413.204,168.340,41.313,157.711
C03353=1033.146,-15.732,413.189,168.343,41.312,157.711
C03354=1033.153,-15.483,413.176,168.346,41.311,157.711
C03355=1033.159,-15.232,413.162,168.348,41.310,157.711
C03356=1033.165,-14.983,413.147,168.351,41.310,157.711
C03357=1033.171,-14.734,413.133,168.353,41.309,157.711
C03358=1033.178,-14.484,413.118,168.356,41.308,157.711
C03359=1033.184,-14.235,413.105,168.358,41.308,157.711
C03360=1033.190,-13.984,413.091,168.361,41.307,157.711
C03361=1033.196,-13.735,413.076,168.363,41.306,157.711
C03362=1033.203,-13.485,413.063,168.366,41.305,157.711
C03363=1033.208,-13.236,413.048,168.367,41.304,157.711
C03364=1033.215,-12.987,413.035,168.370,41.304,157.711
C03365=1033.221,-12.738,413.020,168.372,41.303,157.711
C03366=1033.227,-12.487,413.006,168.375,41.302,157.711
C03367=1033.234,-12.239,412.992,168.377,41.302,157.711
C03368=1033.240,-11.988,412.978,168.380,41.301,157.711
C03369=1033.246,-11.740,412.964,168.382,41.300,157.711
C03370=1033.252,-11.489,412.949,168.385,41.299,157.711
C03371=1033.259,-11.240,412.934,168.387,41.299,157.711
C03372=1033.265,-10.991,412.920,168.390,41.298,157.711
C03373=1033.271,-10.741,412.906,168.392,41.297,157.711
C03374=1033.277,-10.492,412.892,168.395,41.296,157.711
C03375=1033.284,-10.242,412.878,168.396,41.295,157.711
C03376=1033.290,-9.992,412.863,168.400,41.295,157.711
C03377=1033.296,-9.743,412.850,168.401,41.294,157.711
C03378=1033.303,-9.493,412.835,168.404,41.293,157.711
C03379=1033.309,-9.244,412.820,168.406,41.293,157.711
C03380=1033.315,-8.994,412.807,168.409,41.292,157.711
C03381=1033.322,-8.745,412.792,168.411,41.291,157.711
C03382=1033.327,-8.495,412.778,168.414,41.290,157.711
C03383=1033.334,-8.246,412.763,168.416,41.290,157.711
C03384=1033.340,-7.997,412.749,168.419,41.289,157.711
C03385=1033.347,-7.747,412.735,168.421,41.288,157.711
C03386=1033.353,-7.497,412.720,168.424,41.287,157.711
C03387=1033.359,-7.248,412.706,168.426,41.286,157.711
C03388=1033.366,-6.998,412.692,168.428,41.286,157.711
C03389=1033.372,-6.749,412.677,168.430,41.285,157.711
C03390=1033.378,-6.500,412.663,168.432,41.284,157.710
C03391=1033.385,-6.250,412.649,168.435,41.284,157.711
C03392=1033.391,-6.000,412.634,168.437,41.283,157.711
C03393=1033.397,-5.751,412.619,168.440,41.282,157.710
C03394=1033.404,-5.502,412.605,168.442,41.282,157.711
C03395=1033.410,-5.252,412.591,168.445,41.281,157.711
C03396=1033.417,-5.002,412.576,168.447,41.280,157.710
C03397=1033.423,-4.753,412.562,168.450,41.279,157.710
C03398=1033.430,-4.504,412.547,168.452,41.278,157.711
C03399=1033.437,-4.220,412.531,168.455,41.277,157.710
C03400=1033.444,-3.937,412.514,168.458,41.276,157.710
C03401=1033.452,-3.653,412.498,168.460,41.275,157.710
C03402=1033.458,-3.370,412.481,168.462,41.275,157.710
C03403=1033.464,-3.121,412.466,168.465,41.274,157.710
C03404=1033.470,-2.871,412.452,168.467,41.274,157.711
C03405=1033.476,-2.621,412.437,168.470,41.273,157.710
C03406=1033.482,-2.372,412.422,168.472,41.273,157.711
C03407=1033.489,-2.123,412.407,168.475,41.272,157.711
C03408=1033.495,-1.873,412.393,168.477,41.271,157.711
C03409=1033.501,-1.624,412.378,168.479,41.270,157.711
C03410=1033.507,-1.375,412.363,168.482,41.270,157.711
C03411=1033.514,-1.125,412.348,168.484,41.269,157.711
C03412=1033.520,-0.875,412.333,168.487,41.269,157.711
C03413=1033.526,-0.626,412.319,168.489,41.268,157.711
C03414=1033.533,-0.377,412.304,168.491,41.268,157.711
C03415=1033.539,-0.127,412.289,168.494,41.267,157.711
C03416=1033.546,0.122,412.274,168.496,41.266,157.711
C03417=1033.551,0.371,412.260,168.499,41.265,157.711
C03418=1033.558,0.621,412.245,168.501,41.265,157.711
C03419=1033.564,0.871,412.230,168.503,41.264,157.711
C03420=1033.571,1.120,412.215,168.506,41.264,157.711
C03421=1033.576,1.369,412.200,168.507,41.263,157.711
C03422=1033.583,1.619,412.185,168.511,41.262,157.711
C03423=1033.589,1.869,412.170,168.512,41.262,157.711
C03424=1033.595,2.118,412.155,168.514,41.261,157.711
C03425=1033.601,2.367,412.141,168.517,41.260,157.711
C03426=1033.607,2.617,412.125,168.519,41.259,157.711
C03427=1033.613,2.867,412.110,168.522,41.259,157.711
C03428=1033.620,3.116,412.095,168.524,41.258,157.711
C03429=1033.626,3.366,412.080,168.526,41.258,157.711
C03430=1033.632,3.615,412.066,168.529,41.257,157.711
C03431=1033.638,3.865,412.051,168.531,41.257,157.711
C03432=1033.645,4.114,412.036,168.534,41.256,157.711
C03433=1033.651,4.364,412.021,168.536,41.255,157.711
C03434=1033.658,4.613,412.005,168.538,41.254,157.711
C03435=1033.664,4.863,411.990,168.541,41.254,157.711
C03436=1033.670,5.112,411.976,168.543,41.253,157.711
C03437=1033.676,5.361,411.961,168.546,41.252,157.711
C03438=1033.683,5.611,411.946,168.548,41.252,157.711
C03439=1033.689,5.861,411.931,168.549,41.251,157.711
C03440=1033.695,6.110,411.916,168.552,41.251,157.711
C03441=1033.702,6.359,411.900,168.554,41.250,157.711
C03442=1033.708,6.609,411.885,168.557,41.249,157.711
C03443=1033.714,6.858,411.871,168.559,41.248,157.711
C03444=1033.721,7.108,411.856,168.561,41.248,157.711
C03445=1033.727,7.357,411.841,168.564,41.247,157.711
C03446=1033.733,7.607,411.826,168.566,41.246,157.711
C03447=1033.740,7.856,411.810,168.569,41.246,157.711
C03448=1033.746,8.106,411.795,168.571,41.245,157.711
C03449=1033.753,8.355,411.781,168.573,41.245,157.711
C03450=1033.759,8.605,411.766,168.576,41.244,157.711
C03451=1033.766,8.854,411.750,168.578,41.243,157.711
C03452=1033.772,9.104,411.735,168.581,41.242,157.711
C03453=1033.778,9.353,411.720,168.583,41.242,157.711
C03454=1033.784,9.602,411.705,168.585,41.241,157.711
C03455=1033.791,9.851,411.690,168.587,41.240,157.711
C03456=1033.797,10.101,411.675,168.589,41.239,157.711
C03457=1033.803,10.351,411.659,168.592,41.239,157.711
C03458=1033.810,10.601,411.644,168.594,41.238,157.711
C03459=1033.816,10.850,411.629,168.596,41.238,157.711
C03460=1033.823,11.099,411.614,168.599,41.237,157.711
C03461=1033.829,11.349,411.599,168.601,41.236,157.711
C03462=1033.836,11.598,411.583,168.604,41.236,157.711
C03463=1033.843,11.884,411.566,168.606,41.235,157.711
C03464=1033.850,12.168,411.549,168.609,41.234,157.711
C03465=1033.857,12.454,411.531,168.612,41.233,157.711
C03466=1033.865,12.739,411.513,168.614,41.232,157.711
C03467=1033.871,12.988,411.499,168.617,41.231,157.711
C03468=1033.878,13.237,411.483,168.619,41.231,157.711
C03469=1033.884,13.487,411.468,168.621,41.230,157.711
C03470=1033.891,13.737,411.453,168.623,41.229,157.711
C03471=1033.897,13.986,411.437,168.625,41.229,157.711
C03472=1033.903,14.236,411.422,168.628,41.228,157.711
C03473=1033.910,14.485,411.406,168.630,41.228,157.711
C03474=1033.916,14.734,411.391,168.632,41.227,157.711
C03475=1033.922,14.984,411.376,168.635,41.226,157.711
C03476=1033.928,15.233,411.360,168.637,41.226,157.711
C03477=1033.935,15.483,411.345,168.639,41.225,157.711
C03478=1033.942,15.732,411.329,168.642,41.225,157.711
C03479=1033.948,15.981,411.313,168.644,41.224,157.711
C03480=1033.954,16.231,411.298,168.646,41.224,157.711
C03481=1033.961,16.480,411.283,168.649,41.223,157.711
C03482=1033.966,16.730,411.267,168.651,41.223,157.711
C03483=1033.973,16.979,411.251,168.653,41.222,157.711
C03484=1033.979,17.229,411.236,168.656,41.221,157.711
C03485=1033.985,17.478,411.220,168.658,41.220,157.711
C03486=1033.992,17.728,411.205,168.660,41.220,157.711
C03487=1033.998,17.977,411.189,168.663,41.219,157.711
C03488=1034.004,18.226,411.173,168.665,41.219,157.711
C03489=1034.011,18.476,411.158,168.666,41.218,157.711
C03490=1034.017,18.725,411.142,168.670,41.218,157.711
C03491=1034.023,18.975,411.127,168.671,41.217,157.711
C03492=1034.030,19.225,411.111,168.673,41.216,157.711
C03493=1034.036,19.474,411.095,168.676,41.215,157.711
C03494=1034.043,19.724,411.080,168.678,41.215,157.711
C03495=1034.049,19.973,411.064,168.680,41.214,157.711
C03496=1034.055,20.222,411.048,168.683,41.214,157.711
C03497=1034.062,20.472,411.033,168.685,41.213,157.711
C03498=1034.068,20.721,411.017,168.687,41.213,157.711
C03499=1034.074,20.970,411.001,168.690,41.212,157.711
C03500=1034.080,21.220,410.986,168.692,41.211,157.711
C03501=1034.087,21.469,410.970,168.694,41.211,157.711
C03502=1034.093,21.718,410.954,168.696,41.210,157.711
C03503=1034.099,21.968,410.939,168.699,41.210,157.711
C03504=1034.105,22.217,410.922,168.701,41.209,157.711
C03505=1034.112,22.466,410.907,168.703,41.209,157.711
C03506=1034.118,22.717,410.890,168.706,41.208,157.711
C03507=1034.125,22.966,410.875,168.708,41.208,157.711
C03508=1034.130,23.216,410.859,168.710,41.207,157.711
C03509=1034.137,23.465,410.843,168.713,41.206,157.711
C03510=1034.143,23.714,410.827,168.715,41.206,157.711
C03511=1034.150,23.963,410.811,168.717,41.205,157.711
C03512=1034.155,24.213,410.796,168.719,41.205,157.711
C03513=1034.162,24.462,410.780,168.721,41.204,157.711
C03514=1034.169,24.712,410.764,168.723,41.204,157.711
C03515=1034.175,24.961,410.748,168.725,41.203,157.711
C03516=1034.181,25.210,410.732,168.728,41.202,157.712
C03517=1034.188,25.460,410.717,168.730,41.201,157.711
C03518=1034.194,25.709,410.700,168.732,41.201,157.712
C03519=1034.200,25.958,410.685,168.735,41.200,157.711
C03520=1034.207,26.208,410.668,168.737,41.200,157.712
C03521=1034.214,26.458,410.652,168.739,41.199,157.711
C03522=1034.220,26.707,410.636,168.741,41.199,157.712
C03523=1034.226,26.956,410.621,168.744,41.198,157.712
C03524=1034.232,27.206,410.605,168.746,41.198,157.712
C03525=1034.238,27.455,410.589,168.748,41.197,157.712
C03526=1034.245,27.705,410.573,168.751,41.196,157.712
C03527=1034.253,27.991,410.554,168.753,41.196,157.712
C03528=1034.260,28.277,410.535,168.756,41.195,157.712
C03529=1034.267,28.564,410.518,168.759,41.195,157.712
C03530=1034.274,28.851,410.498,168.761,41.194,157.712
C03531=1034.280,29.100,410.483,168.763,41.194,157.712
C03532=1034.286,29.349,410.466,168.766,41.193,157.712
C03533=1034.292,29.599,410.450,168.768,41.192,157.712
C03534=1034.298,29.848,410.434,168.770,41.192,157.712
C03535=1034.305,30.098,410.418,168.771,41.191,157.712
C03536=1034.311,30.347,410.402,168.775,41.191,157.712
C03537=1034.317,30.596,410.385,168.777,41.191,157.712
C03538=1034.324,30.845,410.370,168.778,41.190,157.712
C03539=1034.331,31.095,410.353,168.780,41.189,157.712
C03540=1034.337,31.345,410.337,168.783,41.188,157.712
C03541=1034.343,31.594,410.321,168.785,41.188,157.712
C03542=1034.349,31.843,410.305,168.787,41.188,157.712
C03543=1034.355,32.092,410.288,168.790,41.187,157.712
C03544=1034.362,32.342,410.271,168.792,41.187,157.712
C03545=1034.368,32.591,410.255,168.794,41.186,157.712
C03546=1034.375,32.840,410.239,168.796,41.185,157.712
C03547=1034.381,33.090,410.223,168.799,41.185,157.712
C03548=1034.387,33.340,410.206,168.801,41.184,157.712
C03549=1034.393,33.589,410.190,168.803,41.184,157.712
C03550=1034.400,33.838,410.175,168.805,41.183,157.712
C03551=1034.406,34.088,410.158,168.808,41.183,157.712
C03552=1034.413,34.337,410.141,168.810,41.182,157.712
C03553=1034.419,34.586,410.125,168.812,41.182,157.712
C03554=1034.425,34.836,410.108,168.814,41.181,157.712
C03555=1034.432,35.085,410.092,168.817,41.180,157.712
C03556=1034.438,35.335,410.076,168.819,41.180,157.712
C03557=1034.444,35.584,410.060,168.821,41.179,157.712
C03558=1034.451,35.834,410.043,168.823,41.179,157.712
C03559=1034.457,36.083,410.027,168.826,41.178,157.712
C03560=1034.463,36.332,410.011,168.828,41.178,157.712
C03561=1034.470,36.582,409.994,168.830,41.177,157.712
C03562=1034.476,36.831,409.978,168.832,41.176,157.712
C03563=1034.483,37.080,409.961,168.835,41.176,157.712
C03564=1034.489,37.330,409.945,168.836,41.175,157.712
C03565=1034.495,37.579,409.928,168.838,41.175,157.712
C03566=1034.501,37.828,409.912,168.840,41.175,157.712
C03567=1034.508,38.078,409.895,168.843,41.174,157.712
C03568=1034.514,38.327,409.879,168.845,41.174,157.712
C03569=1034.520,38.577,409.862,168.847,41.173,157.712
C03570=1034.527,38.826,409.845,168.849,41.172,157.712
C03571=1034.533,39.075,409.829,168.852,41.172,157.713
C03572=1034.539,39.325,409.813,168.854,41.172,157.713
C03573=1034.546,39.574,409.795,168.856,41.171,157.713
C03574=1034.551,39.823,409.779,168.858,41.171,157.713
C03575=1034.558,40.072,409.762,168.860,41.170,157.713
C03576=1034.564,40.322,409.745,168.863,41.169,157.713
C03577=1034.570,40.572,409.729,168.865,41.169,157.713
C03578=1034.577,40.820,409.712,168.867,41.169,157.713
C03579=1034.583,41.070,409.695,168.869,41.168,157.713
C03580=1034.589,41.320,409.679,168.872,41.168,157.713
C03581=1034.595,41.568,409.662,168.874,41.167,157.713
C03582=1034.602,41.819,409.646,168.876,41.167,157.713
C03583=1034.608,42.067,409.629,168.878,41.166,157.713
C03584=1034.615,42.317,409.612,168.881,41.166,157.713
C03585=1034.621,42.566,409.595,168.883,41.165,157.713
C03586=1034.627,42.815,409.579,168.885,41.165,157.713
C03587=1034.633,43.065,409.562,168.887,41.165,157.713
C03588=1034.639,43.314,409.545,168.889,41.164,157.713
C03589=1034.645,43.565,409.528,168.892,41.163,157.713
C03590=1034.652,43.813,409.511,168.894,41.163,157.713
C03591=1034.658,44.100,409.492,168.896,41.163,157.713
C03592=1034.665,44.386,409.472,168.899,41.162,157.713
C03593=1034.673,44.673,409.453,168.901,41.162,157.713
C03594=1034.680,44.959,409.433,168.904,41.161,157.713
C03595=1034.686,45.208,409.416,168.906,41.161,157.713
C03596=1034.692,45.458,409.399,168.908,41.160,157.713
C03597=1034.698,45.707,409.382,168.910,41.160,157.713
C03598=1034.705,45.956,409.365,168.912,41.160,157.713
C03599=1034.711,46.206,409.348,168.915,41.159,157.713
C03600=1034.717,46.455,409.331,168.917,41.159,157.714
C03601=1034.724,46.704,409.314,168.919,41.158,157.713
C03602=1034.729,46.954,409.298,168.921,41.158,157.714
C03603=1034.735,47.203,409.280,168.923,41.158,157.714
C03604=1034.742,47.452,409.263,168.926,41.157,157.714
C03605=1034.748,47.701,409.247,168.928,41.156,157.714
C03606=1034.754,47.951,409.229,168.930,41.156,157.714
C03607=1034.760,48.200,409.212,168.932,41.156,157.714
C03608=1034.767,48.450,409.195,168.934,41.156,157.714
C03609=1034.773,48.699,409.178,168.937,41.155,157.714
C03610=1034.779,48.948,409.160,168.939,41.154,157.714
C03611=1034.785,49.198,409.144,168.941,41.154,157.714
C03612=1034.791,49.447,409.127,168.943,41.154,157.714
C03613=1034.797,49.696,409.109,168.945,41.153,157.714
C03614=1034.804,49.945,409.092,168.947,41.153,157.714
C03615=1034.810,50.195,409.075,168.950,41.152,157.714
C03616=1034.816,50.444,409.058,168.951,41.151,157.714
C03617=1034.823,50.694,409.040,168.953,41.151,157.714
C03618=1034.829,50.942,409.023,168.956,41.151,157.714
C03619=1034.835,51.192,409.007,168.958,41.151,157.714
C03620=1034.841,51.441,408.989,168.960,41.150,157.714
C03621=1034.848,51.691,408.972,168.962,41.149,157.714
C03622=1034.854,51.940,408.955,168.964,41.149,157.714
C03623=1034.860,52.190,408.938,168.966,41.148,157.714
C03624=1034.867,52.439,408.920,168.968,41.148,157.714
C03625=1034.873,52.688,408.903,168.971,41.148,157.714
C03626=1034.879,52.938,408.885,168.973,41.147,157.714
C03627=1034.885,53.187,408.869,168.975,41.147,157.714
C03628=1034.892,53.437,408.852,168.977,41.146,157.714
C03629=1034.897,53.686,408.834,168.979,41.146,157.714
C03630=1034.904,53.935,408.817,168.982,41.145,157.714
C03631=1034.911,54.184,408.800,168.984,41.145,157.714
C03632=1034.917,54.433,408.782,168.986,41.145,157.715
C03633=1034.923,54.682,408.765,168.988,41.144,157.714
C03634=1034.929,54.932,408.748,168.990,41.143,157.715
C03635=1034.936,55.182,408.731,168.993,41.143,157.715
C03636=1034.942,55.431,408.714,168.995,41.142,157.715
